Yaskawa INFORM job: A_ROOF_UPPER_0614_2_PAINT_20.JBI

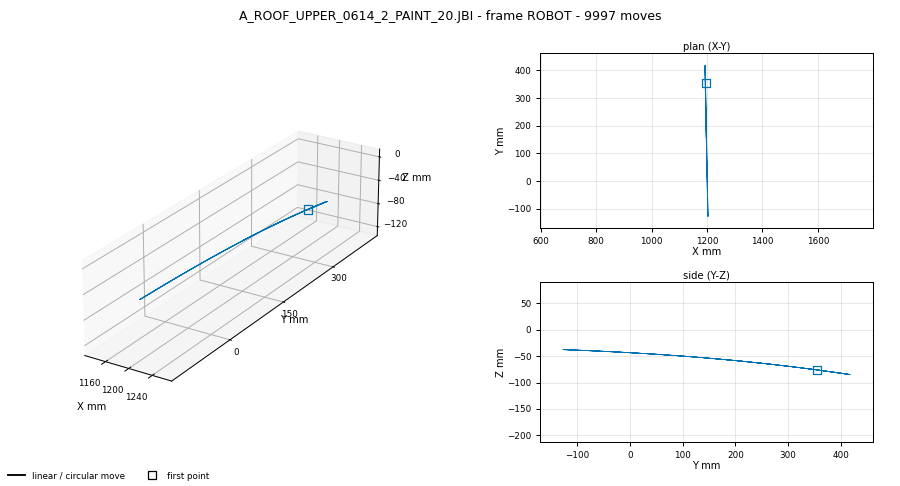
[picture p0: tool path of A_ROOF_UPPER_0614_2_PAINT_20.JBI in frame ROBOT, 9997 of 9997 moves have a stored position in this frame; points joined in program order, loops and branches not executed]
/JOB
//NAME A_ROOF_UPPER_0614_2_PAINT20
//POS
///NPOS 9997,0,0,0,0,0
///TOOL 1
///USER 0
///POSTYPE ROBOT
///RECTAN
///RCONF 1,0,0,0,0,0,0,0,0,0,0,0,0,0,0,0,0,0,0,0,0,0,0,0
C00000=1195.364,354.255,-75.937,-176.133,8.078,148.451
C00001=1195.360,354.502,-75.970,-176.131,8.082,148.451
C00002=1195.356,354.750,-76.004,-176.129,8.085,148.451
C00003=1195.352,354.998,-76.037,-176.128,8.088,148.452
C00004=1195.347,355.246,-76.070,-176.126,8.091,148.452
C00005=1195.343,355.493,-76.103,-176.124,8.095,148.452
C00006=1195.339,355.741,-76.136,-176.122,8.098,148.452
C00007=1195.335,355.989,-76.169,-176.120,8.101,148.453
C00008=1195.331,356.236,-76.203,-176.118,8.104,148.453
C00009=1195.327,356.484,-76.236,-176.116,8.107,148.453
C00010=1195.323,356.732,-76.269,-176.114,8.111,148.454
C00011=1195.319,356.980,-76.302,-176.112,8.114,148.454
C00012=1195.315,357.227,-76.336,-176.110,8.117,148.454
C00013=1195.310,357.475,-76.370,-176.108,8.121,148.455
C00014=1195.306,357.723,-76.403,-176.106,8.124,148.455
C00015=1195.302,357.971,-76.436,-176.105,8.127,148.455
C00016=1195.298,358.219,-76.469,-176.103,8.130,148.455
C00017=1195.294,358.466,-76.503,-176.101,8.134,148.456
C00018=1195.290,358.713,-76.537,-176.099,8.137,148.456
C00019=1195.286,358.961,-76.570,-176.097,8.140,148.456
C00020=1195.282,359.210,-76.603,-176.095,8.143,148.457
C00021=1195.278,359.457,-76.636,-176.093,8.147,148.457
C00022=1195.274,359.705,-76.671,-176.091,8.150,148.457
C00023=1195.269,359.953,-76.704,-176.090,8.153,148.458
C00024=1195.265,360.200,-76.737,-176.088,8.156,148.458
C00025=1195.261,360.448,-76.770,-176.086,8.160,148.458
C00026=1195.258,360.696,-76.805,-176.084,8.163,148.459
C00027=1195.254,360.944,-76.838,-176.082,8.166,148.459
C00028=1195.249,361.192,-76.871,-176.081,8.170,148.459
C00029=1195.245,361.439,-76.905,-176.078,8.173,148.460
C00030=1195.241,361.686,-76.938,-176.077,8.176,148.460
C00031=1195.237,361.934,-76.972,-176.075,8.179,148.460
C00032=1195.234,362.182,-77.006,-176.073,8.183,148.461
C00033=1195.229,362.430,-77.040,-176.072,8.186,148.461
C00034=1195.225,362.677,-77.073,-176.070,8.189,148.461
C00035=1195.221,362.925,-77.107,-176.068,8.193,148.462
C00036=1195.217,363.173,-77.140,-176.067,8.195,148.462
C00037=1195.213,363.420,-77.174,-176.065,8.199,148.463
C00038=1195.208,363.668,-77.208,-176.063,8.202,148.463
C00039=1195.205,363.916,-77.242,-176.061,8.205,148.463
C00040=1195.201,364.163,-77.275,-176.060,8.209,148.464
C00041=1195.196,364.411,-77.309,-176.058,8.212,148.464
C00042=1195.192,364.659,-77.343,-176.056,8.215,148.464
C00043=1195.189,364.906,-77.377,-176.054,8.219,148.465
C00044=1195.184,365.154,-77.410,-176.053,8.221,148.465
C00045=1195.180,365.401,-77.444,-176.051,8.225,148.465
C00046=1195.176,365.650,-77.478,-176.050,8.229,148.466
C00047=1195.172,365.897,-77.512,-176.048,8.231,148.466
C00048=1195.167,366.178,-77.549,-176.047,8.235,148.467
C00049=1195.163,366.459,-77.588,-176.045,8.239,148.467
C00050=1195.159,366.740,-77.627,-176.043,8.242,148.468
C00051=1195.154,367.021,-77.665,-176.041,8.246,148.468
C00052=1195.150,367.268,-77.698,-176.039,8.250,148.468
C00053=1195.146,367.517,-77.733,-176.037,8.253,148.469
C00054=1195.142,367.764,-77.767,-176.036,8.256,148.469
C00055=1195.137,368.012,-77.801,-176.034,8.259,148.470
C00056=1195.133,368.259,-77.835,-176.033,8.262,148.470
C00057=1195.130,368.507,-77.869,-176.031,8.266,148.470
C00058=1195.125,368.755,-77.903,-176.030,8.269,148.471
C00059=1195.121,369.002,-77.937,-176.028,8.272,148.471
C00060=1195.117,369.250,-77.971,-176.027,8.275,148.472
C00061=1195.113,369.498,-78.005,-176.025,8.279,148.472
C00062=1195.109,369.745,-78.038,-176.024,8.282,148.473
C00063=1195.105,369.993,-78.073,-176.023,8.285,148.473
C00064=1195.101,370.241,-78.106,-176.021,8.288,148.473
C00065=1195.097,370.488,-78.141,-176.020,8.292,148.474
C00066=1195.093,370.735,-78.175,-176.018,8.295,148.474
C00067=1195.089,370.983,-78.210,-176.017,8.297,148.475
C00068=1195.085,371.231,-78.243,-176.015,8.301,148.475
C00069=1195.080,371.478,-78.277,-176.014,8.304,148.475
C00070=1195.077,371.726,-78.312,-176.012,8.307,148.476
C00071=1195.073,371.973,-78.345,-176.012,8.311,148.476
C00072=1195.069,372.221,-78.380,-176.010,8.314,148.477
C00073=1195.065,372.469,-78.413,-176.009,8.317,148.477
C00074=1195.060,372.717,-78.448,-176.007,8.320,148.478
C00075=1195.057,372.964,-78.482,-176.005,8.323,148.478
C00076=1195.053,373.212,-78.517,-176.005,8.327,148.479
C00077=1195.048,373.459,-78.551,-176.003,8.329,148.479
C00078=1195.045,373.707,-78.585,-176.002,8.333,148.480
C00079=1195.040,373.955,-78.619,-176.001,8.336,148.480
C00080=1195.036,374.202,-78.653,-175.999,8.340,148.481
C00081=1195.032,374.450,-78.688,-175.998,8.343,148.481
C00082=1195.028,374.697,-78.722,-175.997,8.345,148.481
C00083=1195.024,374.945,-78.756,-175.996,8.348,148.482
C00084=1195.020,375.193,-78.790,-175.994,8.352,148.482
C00085=1195.016,375.440,-78.825,-175.993,8.355,148.483
C00086=1195.013,375.688,-78.859,-175.992,8.358,148.483
C00087=1195.008,375.935,-78.893,-175.990,8.362,148.484
C00088=1195.004,376.183,-78.928,-175.989,8.365,148.484
C00089=1195.000,376.430,-78.962,-175.988,8.367,148.485
C00090=1194.996,376.678,-78.997,-175.987,8.370,148.485
C00091=1194.992,376.926,-79.031,-175.986,8.374,148.486
C00092=1194.988,377.173,-79.065,-175.984,8.377,148.486
C00093=1194.984,377.421,-79.100,-175.984,8.380,148.487
C00094=1194.980,377.668,-79.134,-175.982,8.383,148.487
C00095=1194.976,377.916,-79.168,-175.981,8.387,148.488
C00096=1194.972,378.164,-79.203,-175.980,8.390,148.488
C00097=1194.968,378.411,-79.237,-175.979,8.393,148.489
C00098=1194.964,378.659,-79.272,-175.978,8.396,148.489
C00099=1194.960,378.906,-79.306,-175.977,8.399,148.490
C00100=1194.956,379.154,-79.341,-175.976,8.401,148.490
C00101=1194.951,379.402,-79.375,-175.974,8.405,148.491
C00102=1194.948,379.650,-79.409,-175.973,8.408,148.491
C00103=1194.944,379.897,-79.444,-175.972,8.411,148.492
C00104=1194.939,380.144,-79.478,-175.972,8.414,148.492
C00105=1194.935,380.393,-79.513,-175.970,8.417,148.493
C00106=1194.932,380.639,-79.548,-175.970,8.420,148.493
C00107=1194.928,380.887,-79.583,-175.968,8.423,148.494
C00108=1194.923,381.135,-79.617,-175.968,8.426,148.494
C00109=1194.920,381.382,-79.651,-175.967,8.429,148.495
C00110=1194.915,381.630,-79.686,-175.966,8.432,148.495
C00111=1194.911,381.878,-79.721,-175.965,8.435,148.496
C00112=1194.907,382.125,-79.755,-175.964,8.438,148.496
C00113=1194.904,382.373,-79.790,-175.963,8.441,148.497
C00114=1194.899,382.620,-79.825,-175.962,8.444,148.497
C00115=1194.895,382.868,-79.859,-175.961,8.447,148.498
C00116=1194.891,383.115,-79.893,-175.960,8.450,148.499
C00117=1194.887,383.363,-79.928,-175.959,8.453,148.499
C00118=1194.883,383.610,-79.963,-175.958,8.456,148.500
C00119=1194.879,383.858,-79.998,-175.958,8.459,148.500
C00120=1194.875,384.105,-80.032,-175.957,8.463,148.501
C00121=1194.871,384.353,-80.067,-175.956,8.465,148.501
C00122=1194.867,384.600,-80.102,-175.955,8.468,148.502
C00123=1194.863,384.848,-80.137,-175.954,8.472,148.502
C00124=1194.859,385.096,-80.171,-175.953,8.475,148.503
C00125=1194.855,385.344,-80.205,-175.953,8.477,148.503
C00126=1194.851,385.590,-80.241,-175.952,8.480,148.504
C00127=1194.847,385.839,-80.275,-175.951,8.483,148.504
C00128=1194.843,386.086,-80.310,-175.950,8.486,148.505
C00129=1194.839,386.333,-80.346,-175.949,8.489,148.506
C00130=1194.835,386.581,-80.379,-175.949,8.492,148.506
C00131=1194.831,386.829,-80.414,-175.948,8.494,148.507
C00132=1194.827,387.075,-80.449,-175.948,8.497,148.507
C00133=1194.823,387.324,-80.484,-175.947,8.501,148.508
C00134=1194.819,387.572,-80.519,-175.946,8.503,148.508
C00135=1194.815,387.819,-80.554,-175.945,8.506,148.509
C00136=1194.811,388.066,-80.588,-175.945,8.509,148.509
C00137=1194.807,388.314,-80.623,-175.944,8.512,148.510
C00138=1194.803,388.561,-80.658,-175.943,8.515,148.511
C00139=1194.799,388.809,-80.693,-175.943,8.517,148.511
C00140=1194.795,389.056,-80.729,-175.942,8.520,148.512
C00141=1194.790,389.304,-80.763,-175.941,8.523,148.512
C00142=1194.787,389.551,-80.797,-175.941,8.526,148.513
C00143=1194.783,389.799,-80.833,-175.940,8.529,148.513
C00144=1194.779,390.046,-80.867,-175.940,8.531,148.514
C00145=1194.775,390.294,-80.903,-175.939,8.534,148.514
C00146=1194.771,390.541,-80.937,-175.938,8.537,148.515
C00147=1194.767,390.789,-80.973,-175.938,8.539,148.516
C00148=1194.762,391.036,-81.007,-175.937,8.543,148.516
C00149=1194.758,391.284,-81.042,-175.937,8.545,148.517
C00150=1194.755,391.532,-81.078,-175.936,8.548,148.517
C00151=1194.751,391.779,-81.112,-175.936,8.550,148.518
C00152=1194.747,392.062,-81.152,-175.935,8.553,148.518
C00153=1194.741,392.346,-81.192,-175.934,8.556,148.519
C00154=1194.738,392.629,-81.232,-175.934,8.560,148.520
C00155=1194.732,392.912,-81.272,-175.933,8.563,148.520
C00156=1194.729,393.159,-81.307,-175.933,8.565,148.521
C00157=1194.724,393.407,-81.342,-175.932,8.568,148.522
C00158=1194.720,393.654,-81.377,-175.932,8.571,148.522
C00159=1194.717,393.902,-81.413,-175.931,8.574,148.523
C00160=1194.713,394.149,-81.447,-175.931,8.576,148.523
C00161=1194.709,394.396,-81.482,-175.930,8.579,148.524
C00162=1194.705,394.645,-81.517,-175.930,8.581,148.524
C00163=1194.701,394.891,-81.552,-175.930,8.584,148.525
C00164=1194.697,395.139,-81.587,-175.929,8.587,148.526
C00165=1194.693,395.386,-81.622,-175.929,8.589,148.526
C00166=1194.689,395.634,-81.657,-175.928,8.592,148.527
C00167=1194.685,395.882,-81.693,-175.928,8.595,148.527
C00168=1194.681,396.129,-81.728,-175.928,8.597,148.528
C00169=1194.677,396.377,-81.763,-175.927,8.600,148.528
C00170=1194.673,396.624,-81.798,-175.927,8.602,148.529
C00171=1194.669,396.872,-81.833,-175.927,8.604,148.529
C00172=1194.665,397.119,-81.868,-175.926,8.608,148.530
C00173=1194.661,397.366,-81.904,-175.926,8.610,148.531
C00174=1194.657,397.614,-81.938,-175.925,8.612,148.531
C00175=1194.653,397.862,-81.974,-175.925,8.615,148.532
C00176=1194.648,398.109,-82.008,-175.924,8.617,148.532
C00177=1194.645,398.357,-82.044,-175.924,8.620,148.533
C00178=1194.641,398.604,-82.080,-175.924,8.622,148.533
C00179=1194.637,398.851,-82.114,-175.924,8.625,148.534
C00180=1194.633,399.099,-82.150,-175.923,8.628,148.535
C00181=1194.629,399.346,-82.185,-175.923,8.630,148.535
C00182=1194.625,399.594,-82.220,-175.923,8.632,148.536
C00183=1194.621,399.841,-82.255,-175.923,8.635,148.536
C00184=1194.617,400.089,-82.291,-175.922,8.638,148.537
C00185=1194.613,400.336,-82.325,-175.922,8.640,148.537
C00186=1194.609,400.584,-82.361,-175.921,8.642,148.538
C00187=1194.605,400.831,-82.396,-175.921,8.644,148.538
C00188=1194.601,401.079,-82.431,-175.921,8.647,148.539
C00189=1194.596,401.327,-82.467,-175.921,8.649,148.539
C00190=1194.593,401.574,-82.502,-175.920,8.652,148.540
C00191=1194.588,401.821,-82.537,-175.920,8.655,148.541
C00192=1194.585,402.069,-82.572,-175.920,8.657,148.541
C00193=1194.581,402.316,-82.608,-175.920,8.659,148.542
C00194=1194.577,402.563,-82.643,-175.919,8.661,148.542
C00195=1194.573,402.811,-82.678,-175.919,8.664,148.543
C00196=1194.569,403.059,-82.713,-175.919,8.666,148.543
C00197=1194.565,403.306,-82.749,-175.919,8.668,148.544
C00198=1194.561,403.553,-82.784,-175.918,8.670,148.544
C00199=1194.557,403.801,-82.819,-175.918,8.673,148.545
C00200=1194.553,404.048,-82.854,-175.917,8.676,148.545
C00201=1194.549,404.296,-82.890,-175.917,8.678,148.546
C00202=1194.546,404.543,-82.925,-175.917,8.680,148.547
C00203=1194.541,404.792,-82.961,-175.917,8.683,148.547
C00204=1194.537,405.038,-82.996,-175.917,8.685,148.548
C00205=1194.533,405.286,-83.031,-175.917,8.687,148.548
C00206=1194.529,405.533,-83.067,-175.916,8.690,148.549
C00207=1194.525,405.781,-83.101,-175.916,8.692,148.549
C00208=1194.521,406.028,-83.137,-175.916,8.694,148.550
C00209=1194.517,406.276,-83.173,-175.916,8.697,148.550
C00210=1194.513,406.523,-83.208,-175.915,8.699,148.551
C00211=1194.509,406.770,-83.243,-175.915,8.701,148.551
C00212=1194.505,407.019,-83.279,-175.915,8.703,148.552
C00213=1194.501,407.266,-83.314,-175.915,8.706,148.553
C00214=1194.497,407.513,-83.349,-175.914,8.708,148.553
C00215=1194.493,407.760,-83.385,-175.914,8.710,148.554
C00216=1194.489,408.008,-83.421,-175.914,8.712,148.554
C00217=1194.485,408.255,-83.456,-175.914,8.714,148.555
C00218=1194.481,408.503,-83.491,-175.914,8.716,148.555
C00219=1194.478,408.750,-83.526,-175.914,8.718,148.556
C00220=1194.473,408.998,-83.562,-175.913,8.721,148.556
C00221=1194.469,409.245,-83.597,-175.913,8.723,148.557
C00222=1194.465,409.492,-83.633,-175.913,8.725,148.557
C00223=1194.462,409.740,-83.669,-175.913,8.727,148.558
C00224=1194.458,409.987,-83.704,-175.913,8.730,148.558
C00225=1194.453,410.235,-83.739,-175.912,8.732,148.559
C00226=1194.450,410.482,-83.774,-175.913,8.733,148.559
C00227=1194.445,410.730,-83.810,-175.912,8.736,148.560
C00228=1194.442,410.978,-83.846,-175.912,8.738,148.560
C00229=1194.437,411.224,-83.881,-175.912,8.740,148.561
C00230=1194.434,411.472,-83.917,-175.912,8.742,148.561
C00231=1194.430,411.719,-83.952,-175.911,8.745,148.562
C00232=1194.426,411.967,-83.988,-175.911,8.747,148.562
C00233=1194.421,412.214,-84.023,-175.911,8.748,148.563
C00234=1194.418,412.461,-84.059,-175.911,8.751,148.563
C00235=1194.414,412.710,-84.094,-175.911,8.753,148.564
C00236=1194.410,412.957,-84.129,-175.911,8.755,148.564
C00237=1194.406,413.204,-84.165,-175.910,8.757,148.565
C00238=1194.401,413.452,-84.201,-175.910,8.760,148.566
C00239=1194.398,413.699,-84.236,-175.911,8.761,148.566
C00240=1194.394,413.947,-84.272,-175.910,8.763,148.567
C00241=1194.390,414.194,-84.307,-175.910,8.766,148.567
C00242=1194.386,414.441,-84.342,-175.910,8.768,148.568
C00243=1194.382,414.689,-84.379,-175.910,8.769,148.568
C00244=1194.378,414.936,-84.414,-175.909,8.771,148.568
C00245=1194.374,415.183,-84.449,-175.909,8.774,148.569
C00246=1194.370,415.431,-84.485,-175.909,8.776,148.569
C00247=1194.367,415.678,-84.520,-175.909,8.778,148.570
C00248=1194.360,416.037,-84.572,-175.909,8.781,148.571
C00249=1194.357,416.395,-84.624,-175.909,8.784,148.571
C00250=1194.356,416.753,-84.674,-175.908,8.786,148.572
C00251=1194.359,417.111,-84.725,-175.908,8.789,148.573
C00252=1193.937,417.112,-84.765,-175.912,8.800,148.576
C00253=1193.935,416.751,-84.714,-175.911,8.797,148.576
C00254=1193.935,416.390,-84.662,-175.912,8.795,148.575
C00255=1193.939,416.028,-84.610,-175.912,8.791,148.574
C00256=1193.945,415.668,-84.558,-175.912,8.789,148.574
C00257=1193.949,415.420,-84.523,-175.912,8.787,148.573
C00258=1193.952,415.173,-84.487,-175.912,8.784,148.573
C00259=1193.956,414.925,-84.452,-175.913,8.782,148.572
C00260=1193.961,414.678,-84.416,-175.912,8.781,148.572
C00261=1193.965,414.431,-84.381,-175.913,8.779,148.571
C00262=1193.968,414.183,-84.345,-175.913,8.776,148.571
C00263=1193.972,413.935,-84.310,-175.913,8.774,148.570
C00264=1193.976,413.688,-84.275,-175.914,8.772,148.570
C00265=1193.981,413.440,-84.239,-175.913,8.770,148.569
C00266=1193.985,413.193,-84.203,-175.914,8.768,148.569
C00267=1193.988,412.945,-84.168,-175.914,8.766,148.568
C00268=1193.992,412.698,-84.132,-175.914,8.764,148.568
C00269=1193.996,412.451,-84.097,-175.914,8.761,148.567
C00270=1194.001,412.203,-84.061,-175.914,8.760,148.567
C00271=1194.004,411.956,-84.025,-175.914,8.758,148.566
C00272=1194.008,411.708,-83.990,-175.915,8.755,148.566
C00273=1194.012,411.462,-83.955,-175.915,8.753,148.565
C00274=1194.016,411.214,-83.919,-175.915,8.751,148.565
C00275=1194.020,410.966,-83.883,-175.915,8.749,148.564
C00276=1194.024,410.718,-83.848,-175.915,8.746,148.563
C00277=1194.028,410.471,-83.813,-175.915,8.745,148.563
C00278=1194.032,410.224,-83.777,-175.915,8.743,148.562
C00279=1194.036,409.976,-83.742,-175.916,8.740,148.562
C00280=1194.039,409.729,-83.706,-175.916,8.738,148.561
C00281=1194.044,409.482,-83.670,-175.916,8.736,148.561
C00282=1194.048,409.234,-83.635,-175.916,8.734,148.560
C00283=1194.052,408.987,-83.599,-175.917,8.731,148.560
C00284=1194.055,408.739,-83.564,-175.917,8.729,148.559
C00285=1194.060,408.492,-83.529,-175.917,8.728,148.559
C00286=1194.064,408.244,-83.494,-175.917,8.725,148.558
C00287=1194.067,407.997,-83.458,-175.917,8.723,148.558
C00288=1194.072,407.750,-83.422,-175.917,8.721,148.557
C00289=1194.076,407.502,-83.387,-175.918,8.719,148.557
C00290=1194.080,407.255,-83.351,-175.918,8.716,148.556
C00291=1194.084,407.007,-83.317,-175.918,8.714,148.556
C00292=1194.088,406.760,-83.281,-175.918,8.712,148.555
C00293=1194.091,406.512,-83.246,-175.918,8.709,148.555
C00294=1194.095,406.265,-83.210,-175.918,8.707,148.554
C00295=1194.099,406.018,-83.175,-175.919,8.705,148.553
C00296=1194.104,405.770,-83.139,-175.919,8.702,148.553
C00297=1194.108,405.522,-83.104,-175.919,8.700,148.552
C00298=1194.111,405.274,-83.069,-175.919,8.698,148.552
C00299=1194.116,405.028,-83.033,-175.919,8.696,148.551
C00300=1194.119,404.780,-82.998,-175.920,8.693,148.551
C00301=1194.123,404.532,-82.963,-175.920,8.691,148.550
C00302=1194.128,404.285,-82.928,-175.920,8.689,148.550
C00303=1194.131,404.038,-82.892,-175.920,8.686,148.549
C00304=1194.135,403.790,-82.857,-175.921,8.684,148.549
C00305=1194.139,403.543,-82.821,-175.921,8.682,148.548
C00306=1194.144,403.295,-82.786,-175.921,8.680,148.548
C00307=1194.148,403.048,-82.751,-175.921,8.677,148.547
C00308=1194.151,402.800,-82.715,-175.921,8.675,148.546
C00309=1194.156,402.553,-82.680,-175.922,8.672,148.546
C00310=1194.159,402.305,-82.645,-175.922,8.669,148.545
C00311=1194.163,402.058,-82.609,-175.922,8.667,148.545
C00312=1194.167,401.811,-82.574,-175.923,8.665,148.544
C00313=1194.171,401.563,-82.539,-175.923,8.663,148.544
C00314=1194.175,401.315,-82.504,-175.923,8.660,148.543
C00315=1194.179,401.068,-82.469,-175.923,8.658,148.543
C00316=1194.183,400.821,-82.433,-175.924,8.656,148.542
C00317=1194.187,400.573,-82.398,-175.924,8.653,148.541
C00318=1194.191,400.326,-82.363,-175.925,8.651,148.541
C00319=1194.195,400.078,-82.328,-175.925,8.648,148.540
C00320=1194.199,399.830,-82.293,-175.925,8.646,148.540
C00321=1194.203,399.584,-82.258,-175.925,8.643,148.539
C00322=1194.207,399.336,-82.222,-175.926,8.640,148.539
C00323=1194.211,399.088,-82.187,-175.926,8.638,148.538
C00324=1194.215,398.841,-82.152,-175.926,8.636,148.537
C00325=1194.219,398.593,-82.116,-175.927,8.634,148.537
C00326=1194.223,398.345,-82.081,-175.927,8.630,148.536
C00327=1194.228,398.098,-82.046,-175.928,8.628,148.536
C00328=1194.231,397.851,-82.010,-175.928,8.626,148.535
C00329=1194.235,397.603,-81.975,-175.928,8.623,148.535
C00330=1194.240,397.356,-81.940,-175.928,8.620,148.534
C00331=1194.243,397.108,-81.905,-175.929,8.618,148.533
C00332=1194.248,396.861,-81.870,-175.929,8.616,148.533
C00333=1194.251,396.614,-81.835,-175.930,8.613,148.532
C00334=1194.255,396.365,-81.800,-175.930,8.610,148.532
C00335=1194.260,396.119,-81.765,-175.930,8.608,148.531
C00336=1194.264,395.871,-81.730,-175.931,8.605,148.531
C00337=1194.267,395.623,-81.694,-175.931,8.603,148.530
C00338=1194.272,395.376,-81.659,-175.931,8.600,148.530
C00339=1194.275,395.128,-81.624,-175.932,8.597,148.529
C00340=1194.278,394.881,-81.589,-175.932,8.595,148.529
C00341=1194.283,394.633,-81.555,-175.932,8.592,148.528
C00342=1194.287,394.386,-81.519,-175.933,8.589,148.527
C00343=1194.291,394.139,-81.485,-175.933,8.587,148.527
C00344=1194.295,393.891,-81.449,-175.934,8.584,148.526
C00345=1194.299,393.644,-81.414,-175.934,8.582,148.526
C00346=1194.303,393.396,-81.379,-175.935,8.579,148.525
C00347=1194.307,393.149,-81.344,-175.935,8.576,148.524
C00348=1194.311,392.901,-81.309,-175.936,8.573,148.524
C00349=1194.316,392.618,-81.269,-175.936,8.571,148.523
C00350=1194.320,392.334,-81.229,-175.937,8.568,148.523
C00351=1194.325,392.052,-81.189,-175.937,8.565,148.522
C00352=1194.330,391.768,-81.149,-175.938,8.561,148.521
C00353=1194.333,391.521,-81.114,-175.939,8.558,148.521
C00354=1194.337,391.273,-81.079,-175.939,8.556,148.520
C00355=1194.341,391.026,-81.044,-175.940,8.553,148.520
C00356=1194.345,390.778,-81.009,-175.940,8.551,148.519
C00357=1194.349,390.530,-80.974,-175.941,8.548,148.519
C00358=1194.353,390.283,-80.939,-175.941,8.545,148.518
C00359=1194.357,390.035,-80.904,-175.942,8.542,148.517
C00360=1194.362,389.788,-80.869,-175.943,8.539,148.517
C00361=1194.366,389.540,-80.834,-175.943,8.537,148.516
C00362=1194.369,389.294,-80.800,-175.944,8.534,148.516
C00363=1194.373,389.045,-80.765,-175.945,8.531,148.515
C00364=1194.377,388.798,-80.729,-175.945,8.528,148.515
C00365=1194.381,388.550,-80.695,-175.946,8.525,148.514
C00366=1194.385,388.302,-80.660,-175.947,8.522,148.513
C00367=1194.390,388.056,-80.625,-175.947,8.520,148.513
C00368=1194.394,387.807,-80.590,-175.948,8.517,148.512
C00369=1194.397,387.560,-80.556,-175.948,8.514,148.512
C00370=1194.401,387.313,-80.521,-175.949,8.511,148.511
C00371=1194.405,387.065,-80.486,-175.949,8.508,148.511
C00372=1194.409,386.818,-80.451,-175.950,8.505,148.510
C00373=1194.413,386.570,-80.416,-175.951,8.502,148.510
C00374=1194.418,386.322,-80.381,-175.952,8.499,148.509
C00375=1194.421,386.075,-80.346,-175.953,8.496,148.508
C00376=1194.425,385.828,-80.312,-175.953,8.494,148.508
C00377=1194.429,385.580,-80.277,-175.954,8.491,148.507
C00378=1194.434,385.332,-80.243,-175.955,8.488,148.507
C00379=1194.438,385.085,-80.207,-175.956,8.485,148.506
C00380=1194.441,384.838,-80.173,-175.957,8.482,148.506
C00381=1194.445,384.590,-80.138,-175.958,8.479,148.505
C00382=1194.450,384.343,-80.103,-175.958,8.476,148.505
C00383=1194.454,384.095,-80.068,-175.959,8.473,148.504
C00384=1194.457,383.847,-80.034,-175.959,8.470,148.503
C00385=1194.461,383.599,-80.000,-175.961,8.468,148.503
C00386=1194.466,383.353,-79.964,-175.961,8.464,148.503
C00387=1194.470,383.104,-79.930,-175.962,8.461,148.502
C00388=1194.473,382.857,-79.896,-175.963,8.458,148.501
C00389=1194.477,382.609,-79.861,-175.964,8.455,148.501
C00390=1194.482,382.362,-79.826,-175.965,8.452,148.500
C00391=1194.486,382.114,-79.791,-175.966,8.449,148.500
C00392=1194.489,381.867,-79.757,-175.967,8.446,148.499
C00393=1194.493,381.619,-79.722,-175.968,8.443,148.499
C00394=1194.498,381.372,-79.688,-175.969,8.440,148.498
C00395=1194.502,381.124,-79.653,-175.970,8.437,148.498
C00396=1194.506,380.876,-79.619,-175.971,8.434,148.497
C00397=1194.509,380.629,-79.583,-175.972,8.430,148.497
C00398=1194.514,380.381,-79.549,-175.973,8.428,148.496
C00399=1194.517,380.134,-79.515,-175.974,8.424,148.496
C00400=1194.522,379.886,-79.480,-175.975,8.421,148.495
C00401=1194.526,379.638,-79.445,-175.976,8.419,148.495
C00402=1194.530,379.391,-79.412,-175.977,8.415,148.494
C00403=1194.534,379.144,-79.377,-175.978,8.413,148.494
C00404=1194.538,378.895,-79.342,-175.979,8.410,148.493
C00405=1194.543,378.648,-79.308,-175.981,8.406,148.493
C00406=1194.546,378.400,-79.274,-175.981,8.403,148.492
C00407=1194.550,378.153,-79.238,-175.983,8.400,148.492
C00408=1194.553,377.906,-79.204,-175.983,8.397,148.491
C00409=1194.558,377.658,-79.170,-175.985,8.394,148.491
C00410=1194.563,377.411,-79.135,-175.986,8.390,148.490
C00411=1194.566,377.163,-79.101,-175.987,8.387,148.490
C00412=1194.570,376.916,-79.066,-175.988,8.384,148.489
C00413=1194.574,376.667,-79.032,-175.989,8.381,148.489
C00414=1194.578,376.420,-78.998,-175.990,8.378,148.488
C00415=1194.582,376.172,-78.963,-175.992,8.375,148.488
C00416=1194.586,375.925,-78.929,-175.993,8.372,148.487
C00417=1194.591,375.678,-78.895,-175.994,8.369,148.487
C00418=1194.595,375.430,-78.860,-175.996,8.365,148.486
C00419=1194.599,375.182,-78.827,-175.996,8.362,148.486
C00420=1194.603,374.934,-78.792,-175.998,8.359,148.485
C00421=1194.607,374.687,-78.758,-175.999,8.356,148.485
C00422=1194.611,374.439,-78.723,-176.000,8.353,148.484
C00423=1194.614,374.191,-78.689,-176.001,8.350,148.484
C00424=1194.619,373.944,-78.655,-176.003,8.346,148.483
C00425=1194.622,373.696,-78.621,-176.004,8.343,148.483
C00426=1194.627,373.449,-78.586,-176.005,8.340,148.482
C00427=1194.631,373.202,-78.552,-176.007,8.337,148.482
C00428=1194.634,372.954,-78.517,-176.008,8.334,148.482
C00429=1194.639,372.705,-78.484,-176.009,8.331,148.481
C00430=1194.643,372.458,-78.450,-176.011,8.327,148.481
C00431=1194.647,372.210,-78.415,-176.012,8.324,148.480
C00432=1194.651,371.963,-78.381,-176.014,8.321,148.480
C00433=1194.656,371.716,-78.347,-176.015,8.318,148.479
C00434=1194.659,371.467,-78.313,-176.016,8.315,148.479
C00435=1194.663,371.220,-78.279,-176.018,8.311,148.478
C00436=1194.667,370.973,-78.245,-176.019,8.308,148.478
C00437=1194.671,370.725,-78.210,-176.021,8.305,148.478
C00438=1194.675,370.478,-78.176,-176.022,8.302,148.477
C00439=1194.679,370.230,-78.143,-176.024,8.298,148.477
C00440=1194.683,369.982,-78.108,-176.025,8.295,148.476
C00441=1194.687,369.735,-78.074,-176.027,8.292,148.476
C00442=1194.692,369.487,-78.040,-176.028,8.289,148.476
C00443=1194.695,369.239,-78.006,-176.030,8.285,148.475
C00444=1194.700,368.991,-77.972,-176.031,8.283,148.475
C00445=1194.704,368.744,-77.938,-176.032,8.279,148.474
C00446=1194.707,368.496,-77.904,-176.034,8.276,148.474
C00447=1194.712,368.248,-77.870,-176.035,8.272,148.473
C00448=1194.716,368.001,-77.837,-176.037,8.269,148.473
C00449=1194.721,367.753,-77.802,-176.039,8.266,148.473
C00450=1194.724,367.505,-77.768,-176.040,8.263,148.472
C00451=1194.728,367.258,-77.735,-176.042,8.260,148.472
C00452=1194.733,367.010,-77.700,-176.044,8.256,148.471
C00453=1194.737,366.729,-77.661,-176.045,8.252,148.471
C00454=1194.741,366.448,-77.623,-176.047,8.249,148.470
C00455=1194.746,366.167,-77.585,-176.049,8.245,148.470
C00456=1194.750,365.887,-77.547,-176.051,8.241,148.470
C00457=1194.754,365.639,-77.512,-176.052,8.239,148.469
C00458=1194.759,365.391,-77.479,-176.054,8.235,148.469
C00459=1194.762,365.144,-77.445,-176.056,8.231,148.468
C00460=1194.767,364.896,-77.412,-176.057,8.229,148.468
C00461=1194.770,364.648,-77.377,-176.059,8.225,148.468
C00462=1194.775,364.400,-77.344,-176.060,8.222,148.467
C00463=1194.779,364.153,-77.310,-176.062,8.219,148.467
C00464=1194.783,363.905,-77.277,-176.064,8.215,148.466
C00465=1194.787,363.657,-77.242,-176.065,8.212,148.466
C00466=1194.791,363.410,-77.209,-176.067,8.209,148.466
C00467=1194.795,363.162,-77.175,-176.069,8.205,148.465
C00468=1194.799,362.914,-77.142,-176.070,8.203,148.465
C00469=1194.804,362.667,-77.109,-176.073,8.199,148.465
C00470=1194.807,362.419,-77.074,-176.074,8.196,148.464
C00471=1194.811,362.171,-77.041,-176.076,8.193,148.464
C00472=1194.815,361.924,-77.007,-176.077,8.189,148.464
C00473=1194.820,361.676,-76.974,-176.080,8.186,148.463
C00474=1194.824,361.428,-76.940,-176.081,8.183,148.463
C00475=1194.827,361.180,-76.906,-176.083,8.180,148.463
C00476=1194.831,360.933,-76.873,-176.085,8.176,148.462
C00477=1194.836,360.685,-76.839,-176.087,8.173,148.462
C00478=1194.840,360.438,-76.805,-176.088,8.170,148.462
C00479=1194.844,360.190,-76.772,-176.090,8.166,148.461
C00480=1194.848,359.942,-76.739,-176.092,8.163,148.461
C00481=1194.852,359.694,-76.706,-176.094,8.159,148.461
C00482=1194.855,359.447,-76.672,-176.096,8.157,148.460
C00483=1194.860,359.199,-76.638,-176.098,8.153,148.460
C00484=1194.864,358.951,-76.605,-176.100,8.150,148.460
C00485=1194.869,358.703,-76.572,-176.101,8.147,148.459
C00486=1194.872,358.456,-76.538,-176.103,8.144,148.459
C00487=1194.877,358.208,-76.505,-176.105,8.140,148.459
C00488=1194.880,357.960,-76.471,-176.107,8.137,148.458
C00489=1194.884,357.712,-76.438,-176.109,8.133,148.458
C00490=1194.888,357.464,-76.405,-176.111,8.131,148.458
C00491=1194.892,357.217,-76.371,-176.113,8.127,148.457
C00492=1194.897,356.969,-76.337,-176.115,8.124,148.457
C00493=1194.901,356.721,-76.304,-176.117,8.120,148.457
C00494=1194.905,356.474,-76.271,-176.118,8.118,148.457
C00495=1194.910,356.226,-76.238,-176.120,8.114,148.456
C00496=1194.914,355.978,-76.204,-176.122,8.111,148.456
C00497=1194.918,355.731,-76.171,-176.125,8.107,148.456
C00498=1194.921,355.482,-76.138,-176.126,8.105,148.455
C00499=1194.925,355.234,-76.105,-176.128,8.101,148.455
C00500=1194.930,354.987,-76.071,-176.130,8.098,148.455
C00501=1194.934,354.739,-76.038,-176.132,8.095,148.455
C00502=1194.938,354.492,-76.004,-176.134,8.091,148.454
C00503=1194.942,354.244,-75.971,-176.136,8.088,148.454
C00504=1194.946,353.996,-75.938,-176.138,8.085,148.454
C00505=1194.950,353.749,-75.905,-176.140,8.081,148.453
C00506=1194.954,353.500,-75.873,-176.142,8.078,148.453
C00507=1194.959,353.253,-75.839,-176.144,8.076,148.453
C00508=1194.963,353.005,-75.806,-176.146,8.072,148.453
C00509=1194.967,352.757,-75.773,-176.148,8.069,148.452
C00510=1194.971,352.509,-75.740,-176.150,8.065,148.452
C00511=1194.975,352.262,-75.707,-176.152,8.062,148.452
C00512=1194.979,352.014,-75.674,-176.154,8.059,148.452
C00513=1194.983,351.766,-75.641,-176.156,8.056,148.451
C00514=1194.987,351.519,-75.608,-176.158,8.052,148.451
C00515=1194.991,351.271,-75.575,-176.160,8.049,148.451
C00516=1194.995,351.023,-75.542,-176.162,8.047,148.451
C00517=1195.000,350.775,-75.509,-176.164,8.043,148.450
C00518=1195.004,350.527,-75.476,-176.166,8.040,148.450
C00519=1195.008,350.279,-75.443,-176.168,8.036,148.450
C00520=1195.012,350.032,-75.410,-176.170,8.033,148.449
C00521=1195.016,349.784,-75.377,-176.172,8.031,148.449
C00522=1195.020,349.536,-75.345,-176.174,8.027,148.449
C00523=1195.024,349.288,-75.312,-176.177,8.024,148.449
C00524=1195.028,349.041,-75.278,-176.179,8.021,148.449
C00525=1195.032,348.793,-75.245,-176.181,8.017,148.448
C00526=1195.036,348.545,-75.212,-176.182,8.014,148.448
C00527=1195.041,348.297,-75.180,-176.184,8.011,148.448
C00528=1195.044,348.049,-75.147,-176.187,8.008,148.448
C00529=1195.048,347.802,-75.114,-176.189,8.004,148.447
C00530=1195.053,347.554,-75.082,-176.191,8.002,148.447
C00531=1195.058,347.306,-75.049,-176.193,7.999,148.447
C00532=1195.062,347.058,-75.016,-176.195,7.995,148.447
C00533=1195.065,346.810,-74.984,-176.197,7.992,148.447
C00534=1195.069,346.563,-74.951,-176.200,7.989,148.446
C00535=1195.074,346.315,-74.917,-176.201,7.986,148.446
C00536=1195.078,346.067,-74.885,-176.203,7.983,148.446
C00537=1195.081,345.819,-74.852,-176.206,7.979,148.446
C00538=1195.086,345.571,-74.820,-176.208,7.976,148.445
C00539=1195.090,345.323,-74.787,-176.210,7.973,148.445
C00540=1195.095,345.075,-74.755,-176.212,7.970,148.445
C00541=1195.098,344.828,-74.722,-176.214,7.967,148.445
C00542=1195.103,344.580,-74.689,-176.216,7.964,148.445
C00543=1195.107,344.332,-74.657,-176.219,7.960,148.444
C00544=1195.110,344.085,-74.624,-176.220,7.958,148.444
C00545=1195.115,343.836,-74.592,-176.222,7.954,148.444
C00546=1195.119,343.588,-74.558,-176.225,7.951,148.444
C00547=1195.123,343.341,-74.527,-176.227,7.948,148.444
C00548=1195.128,343.093,-74.494,-176.229,7.944,148.443
C00549=1195.132,342.845,-74.461,-176.231,7.942,148.443
C00550=1195.136,342.597,-74.429,-176.234,7.939,148.443
C00551=1195.140,342.349,-74.396,-176.236,7.936,148.443
C00552=1195.144,342.101,-74.364,-176.238,7.932,148.443
C00553=1195.148,341.854,-74.332,-176.240,7.929,148.443
C00554=1195.153,341.606,-74.299,-176.242,7.926,148.442
C00555=1195.157,341.358,-74.267,-176.244,7.923,148.442
C00556=1195.161,341.110,-74.234,-176.246,7.920,148.442
C00557=1195.165,340.832,-74.198,-176.249,7.916,148.442
C00558=1195.170,340.553,-74.162,-176.251,7.913,148.442
C00559=1195.175,340.275,-74.126,-176.254,7.909,148.441
C00560=1195.179,339.996,-74.089,-176.256,7.906,148.441
C00561=1195.184,339.748,-74.057,-176.259,7.903,148.441
C00562=1195.187,339.500,-74.024,-176.261,7.899,148.441
C00563=1195.192,339.253,-73.992,-176.263,7.897,148.441
C00564=1195.196,339.005,-73.960,-176.265,7.894,148.441
C00565=1195.200,338.756,-73.928,-176.267,7.890,148.440
C00566=1195.204,338.509,-73.895,-176.270,7.887,148.440
C00567=1195.209,338.261,-73.863,-176.271,7.885,148.440
C00568=1195.212,338.013,-73.831,-176.274,7.882,148.440
C00569=1195.217,337.765,-73.799,-176.276,7.878,148.440
C00570=1195.221,337.517,-73.767,-176.279,7.875,148.440
C00571=1195.225,337.270,-73.734,-176.281,7.872,148.439
C00572=1195.229,337.022,-73.702,-176.283,7.869,148.439
C00573=1195.234,336.773,-73.670,-176.285,7.866,148.439
C00574=1195.237,336.525,-73.638,-176.287,7.863,148.439
C00575=1195.242,336.278,-73.606,-176.290,7.859,148.439
C00576=1195.246,336.030,-73.574,-176.292,7.856,148.439
C00577=1195.250,335.781,-73.542,-176.294,7.854,148.439
C00578=1195.254,335.534,-73.509,-176.296,7.851,148.438
C00579=1195.258,335.286,-73.478,-176.298,7.847,148.438
C00580=1195.263,335.038,-73.445,-176.301,7.844,148.438
C00581=1195.266,334.790,-73.413,-176.303,7.842,148.438
C00582=1195.271,334.543,-73.382,-176.305,7.838,148.438
C00583=1195.275,334.294,-73.349,-176.308,7.835,148.438
C00584=1195.279,334.046,-73.318,-176.310,7.832,148.437
C00585=1195.284,333.799,-73.285,-176.312,7.829,148.437
C00586=1195.287,333.551,-73.254,-176.314,7.827,148.437
C00587=1195.291,333.303,-73.222,-176.317,7.823,148.437
C00588=1195.296,333.055,-73.190,-176.319,7.820,148.437
C00589=1195.300,332.807,-73.158,-176.321,7.817,148.437
C00590=1195.304,332.559,-73.126,-176.324,7.814,148.437
C00591=1195.308,332.312,-73.095,-176.325,7.811,148.436
C00592=1195.313,332.063,-73.063,-176.328,7.808,148.436
C00593=1195.317,331.815,-73.031,-176.330,7.805,148.436
C00594=1195.321,331.567,-72.999,-176.333,7.802,148.436
C00595=1195.325,331.319,-72.967,-176.335,7.799,148.436
C00596=1195.329,331.071,-72.936,-176.337,7.796,148.436
C00597=1195.333,330.823,-72.904,-176.340,7.793,148.436
C00598=1195.337,330.575,-72.872,-176.342,7.789,148.436
C00599=1195.342,330.328,-72.840,-176.345,7.786,148.436
C00600=1195.346,330.079,-72.809,-176.346,7.784,148.436
C00601=1195.350,329.832,-72.777,-176.349,7.781,148.436
C00602=1195.354,329.584,-72.745,-176.351,7.778,148.435
C00603=1195.358,329.335,-72.713,-176.353,7.774,148.435
C00604=1195.363,329.087,-72.682,-176.356,7.771,148.435
C00605=1195.367,328.839,-72.650,-176.358,7.769,148.435
C00606=1195.371,328.592,-72.619,-176.360,7.766,148.435
C00607=1195.375,328.344,-72.587,-176.363,7.762,148.435
C00608=1195.380,328.096,-72.556,-176.365,7.759,148.435
C00609=1195.384,327.848,-72.524,-176.367,7.757,148.435
C00610=1195.388,327.600,-72.492,-176.370,7.754,148.435
C00611=1195.392,327.352,-72.461,-176.372,7.751,148.434
C00612=1195.396,327.104,-72.429,-176.375,7.747,148.434
C00613=1195.400,326.856,-72.398,-176.377,7.744,148.434
C00614=1195.404,326.608,-72.367,-176.379,7.742,148.434
C00615=1195.409,326.360,-72.335,-176.381,7.739,148.434
C00616=1195.413,326.112,-72.303,-176.384,7.736,148.434
C00617=1195.417,325.864,-72.272,-176.386,7.732,148.434
C00618=1195.421,325.616,-72.240,-176.388,7.730,148.434
C00619=1195.426,325.368,-72.209,-176.391,7.727,148.434
C00620=1195.430,325.120,-72.178,-176.393,7.724,148.434
C00621=1195.434,324.873,-72.146,-176.395,7.720,148.433
C00622=1195.438,324.624,-72.115,-176.398,7.718,148.433
C00623=1195.442,324.377,-72.083,-176.400,7.715,148.433
C00624=1195.446,324.128,-72.052,-176.403,7.712,148.433
C00625=1195.450,323.881,-72.021,-176.405,7.709,148.433
C00626=1195.454,323.632,-71.990,-176.407,7.706,148.433
C00627=1195.459,323.385,-71.958,-176.410,7.703,148.433
C00628=1195.463,323.136,-71.927,-176.412,7.700,148.433
C00629=1195.467,322.889,-71.896,-176.415,7.697,148.433
C00630=1195.471,322.640,-71.864,-176.417,7.694,148.433
C00631=1195.476,322.392,-71.834,-176.419,7.691,148.433
C00632=1195.479,322.144,-71.802,-176.421,7.688,148.432
C00633=1195.484,321.896,-71.771,-176.424,7.685,148.432
C00634=1195.488,321.649,-71.740,-176.427,7.682,148.432
C00635=1195.492,321.400,-71.709,-176.428,7.680,148.432
C00636=1195.497,321.152,-71.678,-176.431,7.677,148.432
C00637=1195.501,320.904,-71.646,-176.433,7.673,148.432
C00638=1195.505,320.656,-71.615,-176.436,7.670,148.432
C00639=1195.509,320.407,-71.584,-176.439,7.667,148.432
C00640=1195.514,320.160,-71.553,-176.440,7.665,148.432
C00641=1195.518,319.912,-71.522,-176.443,7.662,148.432
C00642=1195.522,319.663,-71.491,-176.446,7.659,148.432
C00643=1195.526,319.416,-71.460,-176.448,7.655,148.432
C00644=1195.530,319.168,-71.429,-176.450,7.653,148.432
C00645=1195.534,318.920,-71.398,-176.453,7.650,148.432
C00646=1195.539,318.672,-71.367,-176.455,7.647,148.432
C00647=1195.543,318.424,-71.335,-176.458,7.644,148.432
C00648=1195.547,318.176,-71.304,-176.460,7.642,148.432
C00649=1195.551,317.927,-71.273,-176.462,7.638,148.431
C00650=1195.556,317.679,-71.243,-176.465,7.635,148.431
C00651=1195.560,317.432,-71.212,-176.467,7.632,148.431
C00652=1195.564,317.184,-71.181,-176.469,7.630,148.431
C00653=1195.568,316.936,-71.150,-176.472,7.627,148.431
C00654=1195.573,316.688,-71.119,-176.474,7.624,148.431
C00655=1195.577,316.439,-71.088,-176.477,7.620,148.431
C00656=1195.581,316.191,-71.058,-176.479,7.618,148.431
C00657=1195.585,315.943,-71.027,-176.482,7.615,148.431
C00658=1195.589,315.695,-70.996,-176.484,7.612,148.431
C00659=1195.594,315.447,-70.965,-176.486,7.609,148.431
C00660=1195.598,315.199,-70.935,-176.489,7.607,148.431
C00661=1195.603,314.922,-70.900,-176.492,7.603,148.431
C00662=1195.607,314.647,-70.865,-176.495,7.600,148.431
C00663=1195.612,314.369,-70.831,-176.497,7.596,148.431
C00664=1195.617,314.094,-70.797,-176.499,7.593,148.431
C00665=1195.621,313.846,-70.766,-176.502,7.590,148.431
C00666=1195.625,313.597,-70.736,-176.505,7.587,148.431
C00667=1195.629,313.349,-70.705,-176.507,7.585,148.431
C00668=1195.634,313.101,-70.674,-176.509,7.582,148.431
C00669=1195.638,312.854,-70.644,-176.512,7.579,148.431
C00670=1195.642,312.605,-70.613,-176.515,7.576,148.431
C00671=1195.646,312.357,-70.582,-176.516,7.573,148.431
C00672=1195.650,312.109,-70.552,-176.519,7.570,148.431
C00673=1195.655,311.861,-70.522,-176.522,7.567,148.431
C00674=1195.659,311.612,-70.491,-176.524,7.565,148.431
C00675=1195.663,311.365,-70.461,-176.527,7.562,148.431
C00676=1195.668,311.117,-70.430,-176.529,7.559,148.430
C00677=1195.672,310.869,-70.399,-176.531,7.556,148.430
C00678=1195.676,310.621,-70.369,-176.534,7.554,148.430
C00679=1195.680,310.372,-70.338,-176.536,7.551,148.430
C00680=1195.684,310.124,-70.309,-176.539,7.548,148.431
C00681=1195.689,309.876,-70.278,-176.541,7.544,148.430
C00682=1195.694,309.628,-70.247,-176.543,7.542,148.430
C00683=1195.697,309.380,-70.216,-176.546,7.539,148.430
C00684=1195.702,309.131,-70.186,-176.549,7.536,148.430
C00685=1195.706,308.884,-70.156,-176.551,7.534,148.430
C00686=1195.710,308.636,-70.125,-176.553,7.531,148.430
C00687=1195.714,308.388,-70.095,-176.556,7.527,148.430
C00688=1195.719,308.139,-70.065,-176.559,7.524,148.430
C00689=1195.722,307.891,-70.035,-176.561,7.522,148.430
C00690=1195.727,307.643,-70.004,-176.563,7.519,148.430
C00691=1195.731,307.395,-69.974,-176.566,7.516,148.430
C00692=1195.736,307.147,-69.944,-176.568,7.513,148.430
C00693=1195.740,306.899,-69.914,-176.570,7.511,148.430
C00694=1195.745,306.651,-69.884,-176.573,7.508,148.430
C00695=1195.748,306.403,-69.853,-176.576,7.505,148.430
C00696=1195.753,306.154,-69.823,-176.578,7.503,148.430
C00697=1195.757,305.906,-69.793,-176.581,7.500,148.430
C00698=1195.761,305.658,-69.762,-176.583,7.497,148.430
C00699=1195.765,305.410,-69.733,-176.586,7.493,148.430
C00700=1195.770,305.162,-69.702,-176.588,7.491,148.430
C00701=1195.774,304.914,-69.672,-176.590,7.488,148.430
C00702=1195.779,304.666,-69.642,-176.593,7.485,148.430
C00703=1195.783,304.417,-69.612,-176.595,7.483,148.430
C00704=1195.787,304.170,-69.582,-176.598,7.480,148.430
C00705=1195.791,303.920,-69.552,-176.601,7.477,148.430
C00706=1195.795,303.673,-69.521,-176.603,7.474,148.430
C00707=1195.800,303.424,-69.491,-176.606,7.472,148.430
C00708=1195.804,303.177,-69.461,-176.608,7.468,148.430
C00709=1195.808,302.928,-69.432,-176.610,7.465,148.430
C00710=1195.813,302.680,-69.402,-176.613,7.463,148.430
C00711=1195.817,302.432,-69.371,-176.615,7.460,148.430
C00712=1195.821,302.184,-69.342,-176.618,7.457,148.430
C00713=1195.826,301.936,-69.311,-176.620,7.455,148.430
C00714=1195.830,301.688,-69.282,-176.623,7.452,148.430
C00715=1195.834,301.439,-69.252,-176.626,7.449,148.430
C00716=1195.839,301.191,-69.222,-176.628,7.447,148.430
C00717=1195.843,300.943,-69.192,-176.630,7.444,148.430
C00718=1195.847,300.695,-69.163,-176.633,7.441,148.431
C00719=1195.851,300.447,-69.133,-176.636,7.438,148.431
C00720=1195.856,300.199,-69.102,-176.638,7.435,148.431
C00721=1195.860,299.950,-69.073,-176.640,7.432,148.430
C00722=1195.864,299.703,-69.043,-176.643,7.429,148.430
C00723=1195.868,299.454,-69.013,-176.645,7.427,148.430
C00724=1195.873,299.206,-68.983,-176.648,7.424,148.430
C00725=1195.877,298.958,-68.954,-176.650,7.421,148.431
C00726=1195.881,298.710,-68.924,-176.653,7.419,148.431
C00727=1195.885,298.462,-68.894,-176.655,7.416,148.431
C00728=1195.890,298.213,-68.864,-176.658,7.413,148.431
C00729=1195.894,297.965,-68.835,-176.660,7.410,148.431
C00730=1195.898,297.717,-68.805,-176.663,7.407,148.431
C00731=1195.903,297.468,-68.776,-176.666,7.404,148.431
C00732=1195.906,297.221,-68.746,-176.668,7.402,148.431
C00733=1195.911,296.972,-68.716,-176.670,7.399,148.431
C00734=1195.916,296.724,-68.686,-176.673,7.396,148.431
C00735=1195.920,296.476,-68.657,-176.675,7.394,148.431
C00736=1195.924,296.227,-68.627,-176.678,7.391,148.431
C00737=1195.928,295.979,-68.598,-176.681,7.388,148.431
C00738=1195.932,295.731,-68.568,-176.683,7.386,148.431
C00739=1195.937,295.482,-68.539,-176.685,7.383,148.431
C00740=1195.941,295.234,-68.509,-176.688,7.380,148.431
C00741=1195.945,294.986,-68.480,-176.690,7.378,148.431
C00742=1195.950,294.738,-68.450,-176.693,7.375,148.431
C00743=1195.955,294.490,-68.421,-176.696,7.372,148.431
C00744=1195.959,294.242,-68.391,-176.698,7.369,148.431
C00745=1195.963,293.993,-68.362,-176.701,7.366,148.431
C00746=1195.967,293.745,-68.333,-176.703,7.363,148.431
C00747=1195.971,293.497,-68.303,-176.705,7.361,148.431
C00748=1195.975,293.248,-68.274,-176.708,7.358,148.431
C00749=1195.980,293.000,-68.244,-176.711,7.355,148.431
C00750=1195.984,292.752,-68.215,-176.713,7.353,148.431
C00751=1195.989,292.504,-68.186,-176.716,7.350,148.431
C00752=1195.993,292.256,-68.156,-176.718,7.347,148.432
C00753=1195.997,292.008,-68.127,-176.721,7.345,148.432
C00754=1196.001,291.760,-68.097,-176.723,7.342,148.432
C00755=1196.005,291.511,-68.068,-176.726,7.339,148.432
C00756=1196.010,291.262,-68.039,-176.729,7.337,148.432
C00757=1196.014,291.014,-68.010,-176.731,7.334,148.432
C00758=1196.019,290.767,-67.981,-176.733,7.332,148.432
C00759=1196.023,290.518,-67.951,-176.736,7.329,148.432
C00760=1196.027,290.270,-67.922,-176.739,7.326,148.432
C00761=1196.032,290.021,-67.893,-176.741,7.324,148.432
C00762=1196.036,289.773,-67.863,-176.744,7.321,148.432
C00763=1196.040,289.526,-67.835,-176.746,7.318,148.432
C00764=1196.044,289.277,-67.805,-176.748,7.315,148.432
C00765=1196.049,289.002,-67.773,-176.751,7.312,148.432
C00766=1196.054,288.728,-67.741,-176.754,7.309,148.432
C00767=1196.058,288.454,-67.709,-176.757,7.307,148.433
C00768=1196.064,288.179,-67.677,-176.760,7.304,148.433
C00769=1196.068,287.931,-67.647,-176.762,7.301,148.433
C00770=1196.071,287.683,-67.618,-176.765,7.298,148.433
C00771=1196.076,287.434,-67.590,-176.767,7.295,148.433
C00772=1196.081,287.187,-67.561,-176.770,7.292,148.433
C00773=1196.085,286.938,-67.532,-176.772,7.290,148.433
C00774=1196.089,286.689,-67.502,-176.775,7.287,148.433
C00775=1196.094,286.441,-67.473,-176.778,7.285,148.433
C00776=1196.098,286.193,-67.445,-176.780,7.282,148.433
C00777=1196.102,285.945,-67.416,-176.783,7.279,148.433
C00778=1196.107,285.696,-67.387,-176.785,7.277,148.433
C00779=1196.111,285.448,-67.357,-176.788,7.274,148.433
C00780=1196.116,285.200,-67.329,-176.790,7.271,148.433
C00781=1196.119,284.952,-67.300,-176.793,7.269,148.433
C00782=1196.124,284.703,-67.271,-176.795,7.266,148.433
C00783=1196.129,284.455,-67.242,-176.797,7.264,148.433
C00784=1196.133,284.207,-67.213,-176.801,7.261,148.434
C00785=1196.137,283.958,-67.185,-176.803,7.258,148.434
C00786=1196.141,283.709,-67.156,-176.805,7.256,148.434
C00787=1196.146,283.462,-67.127,-176.808,7.253,148.434
C00788=1196.150,283.213,-67.098,-176.810,7.251,148.434
C00789=1196.154,282.965,-67.069,-176.813,7.248,148.434
C00790=1196.159,282.717,-67.041,-176.816,7.245,148.434
C00791=1196.163,282.469,-67.012,-176.818,7.243,148.434
C00792=1196.167,282.220,-66.983,-176.821,7.240,148.434
C00793=1196.172,281.972,-66.955,-176.823,7.238,148.434
C00794=1196.176,281.724,-66.926,-176.826,7.235,148.434
C00795=1196.180,281.475,-66.897,-176.829,7.232,148.434
C00796=1196.185,281.227,-66.869,-176.831,7.229,148.435
C00797=1196.189,280.979,-66.840,-176.834,7.227,148.435
C00798=1196.193,280.731,-66.812,-176.836,7.225,148.435
C00799=1196.198,280.482,-66.783,-176.839,7.222,148.435
C00800=1196.202,280.234,-66.754,-176.841,7.219,148.435
C00801=1196.206,279.986,-66.726,-176.844,7.216,148.435
C00802=1196.211,279.737,-66.697,-176.846,7.213,148.435
C00803=1196.214,279.489,-66.668,-176.849,7.212,148.435
C00804=1196.219,279.241,-66.640,-176.852,7.209,148.435
C00805=1196.224,278.992,-66.611,-176.854,7.206,148.435
C00806=1196.228,278.744,-66.583,-176.857,7.203,148.435
C00807=1196.233,278.495,-66.555,-176.859,7.201,148.436
C00808=1196.236,278.247,-66.526,-176.862,7.199,148.436
C00809=1196.241,277.999,-66.497,-176.865,7.196,148.436
C00810=1196.245,277.750,-66.469,-176.867,7.193,148.436
C00811=1196.250,277.502,-66.441,-176.869,7.190,148.436
C00812=1196.254,277.254,-66.413,-176.872,7.188,148.436
C00813=1196.259,277.005,-66.384,-176.875,7.185,148.436
C00814=1196.262,276.757,-66.356,-176.877,7.183,148.436
C00815=1196.267,276.508,-66.327,-176.880,7.180,148.436
C00816=1196.271,276.261,-66.299,-176.882,7.178,148.436
C00817=1196.276,276.012,-66.270,-176.884,7.175,148.436
C00818=1196.280,275.764,-66.242,-176.888,7.172,148.437
C00819=1196.285,275.515,-66.214,-176.890,7.170,148.437
C00820=1196.289,275.267,-66.186,-176.893,7.167,148.437
C00821=1196.293,275.018,-66.157,-176.895,7.165,148.437
C00822=1196.298,274.770,-66.129,-176.898,7.162,148.437
C00823=1196.302,274.521,-66.101,-176.900,7.160,148.437
C00824=1196.307,274.274,-66.073,-176.903,7.157,148.437
C00825=1196.310,274.025,-66.045,-176.905,7.155,148.437
C00826=1196.315,273.777,-66.016,-176.908,7.152,148.437
C00827=1196.319,273.528,-65.988,-176.910,7.150,148.438
C00828=1196.324,273.280,-65.960,-176.913,7.147,148.438
C00829=1196.328,273.031,-65.932,-176.915,7.145,148.438
C00830=1196.332,272.784,-65.904,-176.918,7.142,148.438
C00831=1196.337,272.535,-65.875,-176.921,7.139,148.438
C00832=1196.341,272.287,-65.847,-176.923,7.137,148.438
C00833=1196.345,272.038,-65.819,-176.926,7.134,148.438
C00834=1196.350,271.789,-65.792,-176.928,7.132,148.438
C00835=1196.354,271.541,-65.764,-176.931,7.129,148.439
C00836=1196.358,271.293,-65.736,-176.933,7.127,148.439
C00837=1196.363,271.044,-65.707,-176.936,7.124,148.439
C00838=1196.367,270.796,-65.679,-176.938,7.122,148.439
C00839=1196.372,270.548,-65.651,-176.941,7.119,148.439
C00840=1196.376,270.299,-65.623,-176.943,7.117,148.439
C00841=1196.381,270.051,-65.596,-176.946,7.114,148.439
C00842=1196.385,269.802,-65.568,-176.949,7.112,148.439
C00843=1196.390,269.554,-65.539,-176.951,7.109,148.439
C00844=1196.393,269.306,-65.511,-176.954,7.107,148.440
C00845=1196.398,269.057,-65.484,-176.956,7.104,148.440
C00846=1196.402,268.809,-65.456,-176.959,7.102,148.440
C00847=1196.407,268.560,-65.427,-176.962,7.099,148.440
C00848=1196.412,268.312,-65.400,-176.964,7.097,148.440
C00849=1196.416,268.064,-65.373,-176.967,7.094,148.440
C00850=1196.420,267.815,-65.344,-176.969,7.092,148.440
C00851=1196.425,267.567,-65.317,-176.972,7.089,148.440
C00852=1196.429,267.318,-65.289,-176.974,7.087,148.441
C00853=1196.433,267.070,-65.261,-176.977,7.084,148.441
C00854=1196.438,266.822,-65.234,-176.979,7.082,148.441
C00855=1196.442,266.573,-65.206,-176.982,7.079,148.441
C00856=1196.446,266.325,-65.178,-176.985,7.077,148.441
C00857=1196.451,266.076,-65.150,-176.987,7.074,148.441
C00858=1196.455,265.828,-65.122,-176.990,7.072,148.441
C00859=1196.460,265.579,-65.095,-176.993,7.069,148.442
C00860=1196.464,265.331,-65.067,-176.995,7.067,148.442
C00861=1196.468,265.082,-65.040,-176.998,7.064,148.442
C00862=1196.472,264.834,-65.012,-177.000,7.062,148.442
C00863=1196.477,264.586,-64.985,-177.002,7.060,148.442
C00864=1196.482,264.337,-64.956,-177.005,7.057,148.442
C00865=1196.486,264.088,-64.929,-177.008,7.055,148.442
C00866=1196.491,263.841,-64.901,-177.010,7.052,148.442
C00867=1196.495,263.591,-64.874,-177.013,7.050,148.443
C00868=1196.499,263.344,-64.846,-177.016,7.048,148.443
C00869=1196.504,263.071,-64.816,-177.018,7.045,148.443
C00870=1196.508,262.798,-64.786,-177.021,7.043,148.443
C00871=1196.513,262.525,-64.756,-177.024,7.040,148.443
C00872=1196.519,262.253,-64.725,-177.027,7.037,148.443
C00873=1196.523,262.003,-64.698,-177.029,7.035,148.444
C00874=1196.527,261.755,-64.671,-177.032,7.032,148.444
C00875=1196.532,261.507,-64.643,-177.034,7.030,148.444
C00876=1196.536,261.259,-64.616,-177.037,7.027,148.444
C00877=1196.540,261.010,-64.588,-177.039,7.025,148.444
C00878=1196.545,260.762,-64.561,-177.043,7.022,148.444
C00879=1196.550,260.513,-64.534,-177.045,7.020,148.444
C00880=1196.554,260.265,-64.507,-177.047,7.017,148.444
C00881=1196.558,260.016,-64.478,-177.050,7.015,148.445
C00882=1196.563,259.767,-64.451,-177.052,7.013,148.445
C00883=1196.567,259.519,-64.424,-177.055,7.010,148.445
C00884=1196.572,259.271,-64.396,-177.058,7.008,148.445
C00885=1196.575,259.023,-64.370,-177.060,7.005,148.445
C00886=1196.580,258.774,-64.343,-177.063,7.003,148.446
C00887=1196.584,258.525,-64.316,-177.066,7.000,148.446
C00888=1196.589,258.277,-64.288,-177.068,6.998,148.446
C00889=1196.593,258.029,-64.261,-177.070,6.996,148.446
C00890=1196.598,257.780,-64.234,-177.073,6.993,148.446
C00891=1196.602,257.531,-64.206,-177.076,6.991,148.446
C00892=1196.607,257.283,-64.179,-177.078,6.988,148.446
C00893=1196.611,257.034,-64.152,-177.081,6.986,148.446
C00894=1196.616,256.786,-64.124,-177.084,6.984,148.447
C00895=1196.620,256.538,-64.098,-177.086,6.981,148.447
C00896=1196.624,256.290,-64.071,-177.089,6.980,148.447
C00897=1196.628,256.040,-64.043,-177.091,6.977,148.447
C00898=1196.633,255.792,-64.016,-177.093,6.974,148.447
C00899=1196.638,255.543,-63.989,-177.097,6.972,148.448
C00900=1196.642,255.295,-63.962,-177.099,6.969,148.448
C00901=1196.646,255.047,-63.936,-177.101,6.968,148.448
C00902=1196.651,254.798,-63.909,-177.104,6.965,148.448
C00903=1196.655,254.550,-63.882,-177.106,6.962,148.448
C00904=1196.659,254.301,-63.854,-177.109,6.960,148.448
C00905=1196.664,254.052,-63.827,-177.112,6.958,148.448
C00906=1196.668,253.804,-63.801,-177.114,6.956,148.449
C00907=1196.673,253.555,-63.774,-177.117,6.953,148.449
C00908=1196.677,253.307,-63.747,-177.120,6.951,148.449
C00909=1196.682,253.058,-63.719,-177.122,6.948,148.449
C00910=1196.686,252.810,-63.693,-177.125,6.946,148.450
C00911=1196.691,252.562,-63.666,-177.127,6.944,148.450
C00912=1196.695,252.313,-63.639,-177.130,6.941,148.450
C00913=1196.700,252.065,-63.612,-177.132,6.939,148.450
C00914=1196.704,251.817,-63.585,-177.135,6.937,148.450
C00915=1196.708,251.567,-63.558,-177.138,6.934,148.450
C00916=1196.713,251.319,-63.531,-177.140,6.932,148.450
C00917=1196.716,251.071,-63.504,-177.143,6.929,148.451
C00918=1196.721,250.822,-63.478,-177.145,6.927,148.451
C00919=1196.726,250.573,-63.451,-177.148,6.925,148.451
C00920=1196.730,250.325,-63.425,-177.151,6.922,148.451
C00921=1196.735,250.076,-63.397,-177.153,6.920,148.451
C00922=1196.739,249.828,-63.370,-177.155,6.918,148.452
C00923=1196.743,249.580,-63.344,-177.158,6.915,148.452
C00924=1196.748,249.331,-63.318,-177.161,6.914,148.452
C00925=1196.753,249.082,-63.291,-177.163,6.911,148.452
C00926=1196.757,248.834,-63.264,-177.166,6.909,148.452
C00927=1196.761,248.585,-63.237,-177.168,6.907,148.452
C00928=1196.766,248.337,-63.211,-177.171,6.904,148.453
C00929=1196.770,248.088,-63.184,-177.174,6.902,148.453
C00930=1196.775,247.840,-63.157,-177.176,6.900,148.453
C00931=1196.779,247.591,-63.131,-177.179,6.897,148.453
C00932=1196.784,247.342,-63.104,-177.182,6.895,148.453
C00933=1196.788,247.094,-63.078,-177.184,6.893,148.454
C00934=1196.793,246.845,-63.051,-177.187,6.890,148.454
C00935=1196.797,246.597,-63.025,-177.189,6.888,148.454
C00936=1196.801,246.348,-62.998,-177.192,6.886,148.454
C00937=1196.806,246.100,-62.972,-177.194,6.883,148.454
C00938=1196.810,245.851,-62.945,-177.197,6.881,148.455
C00939=1196.815,245.603,-62.918,-177.199,6.879,148.455
C00940=1196.819,245.354,-62.892,-177.202,6.877,148.455
C00941=1196.824,245.105,-62.865,-177.205,6.874,148.455
C00942=1196.828,244.856,-62.840,-177.207,6.873,148.455
C00943=1196.832,244.608,-62.813,-177.210,6.870,148.455
C00944=1196.837,244.360,-62.786,-177.213,6.868,148.456
C00945=1196.841,244.112,-62.761,-177.215,6.866,148.456
C00946=1196.846,243.863,-62.734,-177.218,6.863,148.456
C00947=1196.850,243.614,-62.708,-177.220,6.861,148.456
C00948=1196.855,243.366,-62.681,-177.223,6.859,148.457
C00949=1196.859,243.117,-62.655,-177.225,6.856,148.457
C00950=1196.864,242.869,-62.628,-177.228,6.854,148.457
C00951=1196.868,242.620,-62.602,-177.230,6.852,148.457
C00952=1196.872,242.371,-62.576,-177.233,6.849,148.457
C00953=1196.877,242.122,-62.549,-177.236,6.847,148.458
C00954=1196.882,241.874,-62.524,-177.238,6.845,148.458
C00955=1196.886,241.626,-62.497,-177.241,6.843,148.458
C00956=1196.891,241.377,-62.471,-177.244,6.840,148.458
C00957=1196.894,241.129,-62.445,-177.246,6.839,148.458
C00958=1196.899,240.880,-62.418,-177.248,6.836,148.459
C00959=1196.904,240.631,-62.393,-177.252,6.834,148.459
C00960=1196.908,240.382,-62.366,-177.254,6.832,148.459
C00961=1196.913,240.134,-62.340,-177.256,6.830,148.459
C00962=1196.917,239.886,-62.314,-177.259,6.827,148.459
C00963=1196.922,239.637,-62.287,-177.262,6.825,148.460
C00964=1196.926,239.388,-62.262,-177.264,6.823,148.460
C00965=1196.931,239.139,-62.236,-177.267,6.820,148.460
C00966=1196.935,238.891,-62.209,-177.270,6.818,148.460
C00967=1196.940,238.643,-62.183,-177.272,6.816,148.460
C00968=1196.944,238.394,-62.158,-177.275,6.814,148.461
C00969=1196.948,238.145,-62.132,-177.277,6.811,148.461
C00970=1196.953,237.897,-62.105,-177.280,6.809,148.461
C00971=1196.957,237.648,-62.079,-177.283,6.808,148.461
C00972=1196.962,237.399,-62.053,-177.285,6.805,148.461
C00973=1196.967,237.129,-62.025,-177.288,6.803,148.462
C00974=1196.972,236.856,-61.996,-177.291,6.800,148.462
C00975=1196.977,236.584,-61.968,-177.293,6.798,148.462
C00976=1196.982,236.314,-61.940,-177.296,6.795,148.462
C00977=1196.986,236.065,-61.914,-177.299,6.793,148.463
C00978=1196.990,235.816,-61.888,-177.301,6.791,148.463
C00979=1196.995,235.567,-61.862,-177.304,6.789,148.463
C00980=1197.000,235.319,-61.837,-177.307,6.786,148.463
C00981=1197.004,235.070,-61.811,-177.309,6.785,148.464
C00982=1197.008,234.822,-61.784,-177.312,6.783,148.464
C00983=1197.012,234.573,-61.759,-177.315,6.780,148.464
C00984=1197.017,234.325,-61.733,-177.317,6.778,148.464
C00985=1197.022,234.076,-61.707,-177.320,6.776,148.465
C00986=1197.026,233.827,-61.681,-177.322,6.774,148.465
C00987=1197.030,233.578,-61.655,-177.325,6.771,148.465
C00988=1197.035,233.330,-61.630,-177.327,6.769,148.465
C00989=1197.040,233.081,-61.604,-177.330,6.767,148.465
C00990=1197.044,232.833,-61.579,-177.333,6.765,148.466
C00991=1197.049,232.585,-61.553,-177.335,6.762,148.466
C00992=1197.053,232.336,-61.527,-177.338,6.761,148.466
C00993=1197.058,232.087,-61.501,-177.340,6.758,148.466
C00994=1197.063,231.839,-61.476,-177.343,6.757,148.467
C00995=1197.067,231.590,-61.450,-177.346,6.754,148.467
C00996=1197.071,231.341,-61.424,-177.348,6.752,148.467
C00997=1197.076,231.093,-61.399,-177.351,6.750,148.467
C00998=1197.080,230.843,-61.374,-177.353,6.748,148.468
C00999=1197.085,230.595,-61.348,-177.356,6.745,148.468
C01000=1197.089,230.346,-61.323,-177.359,6.743,148.468
C01001=1197.094,230.098,-61.297,-177.361,6.741,148.468
C01002=1197.098,229.849,-61.271,-177.364,6.739,148.468
C01003=1197.103,229.601,-61.246,-177.367,6.737,148.469
C01004=1197.107,229.352,-61.220,-177.369,6.735,148.469
C01005=1197.111,229.103,-61.194,-177.372,6.733,148.469
C01006=1197.116,228.854,-61.170,-177.374,6.731,148.470
C01007=1197.121,228.606,-61.144,-177.378,6.728,148.470
C01008=1197.125,228.357,-61.118,-177.380,6.726,148.470
C01009=1197.130,228.109,-61.093,-177.382,6.724,148.470
C01010=1197.134,227.860,-61.067,-177.385,6.722,148.471
C01011=1197.139,227.611,-61.042,-177.387,6.720,148.471
C01012=1197.143,227.362,-61.017,-177.390,6.718,148.471
C01013=1197.147,227.114,-60.991,-177.393,6.716,148.471
C01014=1197.153,226.865,-60.966,-177.395,6.714,148.471
C01015=1197.157,226.616,-60.940,-177.398,6.712,148.472
C01016=1197.162,226.368,-60.915,-177.401,6.709,148.472
C01017=1197.166,226.119,-60.889,-177.403,6.707,148.472
C01018=1197.170,225.870,-60.865,-177.406,6.705,148.472
C01019=1197.174,225.622,-60.839,-177.408,6.703,148.473
C01020=1197.179,225.373,-60.814,-177.411,6.701,148.473
C01021=1197.184,225.124,-60.789,-177.414,6.698,148.473
C01022=1197.188,224.876,-60.763,-177.416,6.697,148.474
C01023=1197.193,224.628,-60.738,-177.419,6.694,148.474
C01024=1197.197,224.378,-60.713,-177.421,6.693,148.474
C01025=1197.202,224.130,-60.687,-177.424,6.691,148.474
C01026=1197.206,223.881,-60.663,-177.427,6.688,148.475
C01027=1197.210,223.632,-60.637,-177.429,6.686,148.475
C01028=1197.215,223.383,-60.613,-177.432,6.684,148.475
C01029=1197.220,223.135,-60.587,-177.435,6.682,148.475
C01030=1197.224,222.886,-60.561,-177.437,6.680,148.475
C01031=1197.229,222.637,-60.536,-177.440,6.678,148.476
C01032=1197.233,222.389,-60.512,-177.443,6.676,148.476
C01033=1197.238,222.140,-60.487,-177.445,6.674,148.476
C01034=1197.242,221.892,-60.461,-177.447,6.672,148.477
C01035=1197.247,221.642,-60.436,-177.450,6.670,148.477
C01036=1197.251,221.394,-60.411,-177.453,6.668,148.477
C01037=1197.256,221.145,-60.386,-177.455,6.665,148.477
C01038=1197.261,220.896,-60.362,-177.458,6.663,148.478
C01039=1197.265,220.648,-60.336,-177.461,6.661,148.478
C01040=1197.269,220.399,-60.312,-177.463,6.660,148.478
C01041=1197.273,220.150,-60.286,-177.465,6.657,148.478
C01042=1197.279,219.902,-60.261,-177.469,6.655,148.479
C01043=1197.283,219.653,-60.236,-177.471,6.653,148.479
C01044=1197.287,219.404,-60.212,-177.474,6.651,148.479
C01045=1197.292,219.156,-60.187,-177.476,6.649,148.479
C01046=1197.297,218.907,-60.161,-177.479,6.647,148.480
C01047=1197.301,218.658,-60.137,-177.481,6.645,148.480
C01048=1197.306,218.409,-60.112,-177.485,6.643,148.480
C01049=1197.310,218.161,-60.087,-177.487,6.641,148.481
C01050=1197.314,217.912,-60.062,-177.489,6.639,148.481
C01051=1197.319,217.663,-60.038,-177.492,6.637,148.481
C01052=1197.324,217.415,-60.012,-177.495,6.635,148.482
C01053=1197.328,217.166,-59.988,-177.497,6.633,148.482
C01054=1197.333,216.917,-59.963,-177.500,6.630,148.482
C01055=1197.337,216.668,-59.939,-177.503,6.628,148.482
C01056=1197.342,216.420,-59.913,-177.505,6.627,148.483
C01057=1197.347,216.171,-59.889,-177.508,6.625,148.483
C01058=1197.351,215.922,-59.864,-177.510,6.623,148.483
C01059=1197.356,215.673,-59.839,-177.513,6.621,148.483
C01060=1197.359,215.424,-59.815,-177.516,6.618,148.484
C01061=1197.364,215.176,-59.790,-177.519,6.616,148.484
C01062=1197.369,214.927,-59.765,-177.521,6.614,148.484
C01063=1197.373,214.678,-59.740,-177.524,6.612,148.484
C01064=1197.378,214.430,-59.716,-177.526,6.611,148.485
C01065=1197.383,214.181,-59.692,-177.529,6.609,148.485
C01066=1197.387,213.932,-59.667,-177.532,6.607,148.485
C01067=1197.391,213.684,-59.642,-177.534,6.604,148.486
C01068=1197.397,213.435,-59.617,-177.537,6.602,148.486
C01069=1197.400,213.186,-59.593,-177.540,6.600,148.486
C01070=1197.405,212.937,-59.568,-177.542,6.598,148.487
C01071=1197.410,212.689,-59.544,-177.545,6.597,148.487
C01072=1197.414,212.440,-59.519,-177.547,6.594,148.487
C01073=1197.419,212.191,-59.495,-177.550,6.593,148.487
C01074=1197.424,211.942,-59.470,-177.553,6.590,148.488
C01075=1197.428,211.693,-59.446,-177.556,6.588,148.488
C01076=1197.433,211.445,-59.421,-177.558,6.586,148.488
C01077=1197.438,211.174,-59.394,-177.561,6.585,148.489
C01078=1197.442,210.905,-59.368,-177.564,6.582,148.489
C01079=1197.447,210.633,-59.342,-177.567,6.580,148.489
C01080=1197.452,210.363,-59.315,-177.569,6.578,148.490
C01081=1197.457,210.114,-59.291,-177.572,6.575,148.490
C01082=1197.461,209.865,-59.266,-177.575,6.573,148.490
C01083=1197.466,209.617,-59.242,-177.577,6.572,148.490
C01084=1197.471,209.368,-59.217,-177.580,6.570,148.491
C01085=1197.475,209.119,-59.193,-177.583,6.568,148.491
C01086=1197.479,208.870,-59.169,-177.585,6.566,148.491
C01087=1197.484,208.622,-59.144,-177.587,6.564,148.492
C01088=1197.489,208.373,-59.120,-177.590,6.562,148.492
C01089=1197.494,208.124,-59.096,-177.593,6.560,148.492
C01090=1197.498,207.875,-59.072,-177.596,6.558,148.493
C01091=1197.502,207.626,-59.048,-177.599,6.556,148.493
C01092=1197.507,207.378,-59.023,-177.601,6.554,148.493
C01093=1197.512,207.129,-58.999,-177.603,6.552,148.493
C01094=1197.516,206.881,-58.975,-177.606,6.550,148.494
C01095=1197.521,206.631,-58.951,-177.609,6.548,148.494
C01096=1197.525,206.382,-58.926,-177.611,6.546,148.494
C01097=1197.530,206.134,-58.902,-177.614,6.545,148.495
C01098=1197.535,205.885,-58.878,-177.617,6.543,148.495
C01099=1197.540,205.636,-58.854,-177.619,6.541,148.495
C01100=1197.543,205.387,-58.830,-177.622,6.538,148.495
C01101=1197.548,205.139,-58.806,-177.625,6.536,148.496
C01102=1197.553,204.890,-58.781,-177.627,6.534,148.496
C01103=1197.558,204.641,-58.758,-177.630,6.533,148.496
C01104=1197.562,204.392,-58.734,-177.633,6.531,148.497
C01105=1197.566,204.144,-58.710,-177.635,6.529,148.497
C01106=1197.571,203.894,-58.685,-177.638,6.527,148.497
C01107=1197.576,203.646,-58.661,-177.640,6.525,148.498
C01108=1197.580,203.397,-58.637,-177.643,6.523,148.498
C01109=1197.585,203.148,-58.614,-177.646,6.521,148.498
C01110=1197.589,202.900,-58.590,-177.648,6.520,148.499
C01111=1197.594,202.651,-58.565,-177.651,6.518,148.499
C01112=1197.598,202.401,-58.541,-177.653,6.516,148.499
C01113=1197.603,202.153,-58.517,-177.656,6.513,148.499
C01114=1197.607,201.904,-58.494,-177.659,6.511,148.500
C01115=1197.612,201.655,-58.470,-177.662,6.509,148.500
C01116=1197.616,201.406,-58.447,-177.664,6.508,148.500
C01117=1197.622,201.158,-58.422,-177.667,6.506,148.501
C01118=1197.626,200.909,-58.398,-177.669,6.504,148.501
C01119=1197.631,200.660,-58.374,-177.672,6.502,148.501
C01120=1197.635,200.412,-58.350,-177.675,6.500,148.502
C01121=1197.639,200.162,-58.327,-177.677,6.498,148.502
C01122=1197.644,199.914,-58.303,-177.680,6.496,148.502
C01123=1197.648,199.665,-58.279,-177.682,6.494,148.503
C01124=1197.653,199.416,-58.255,-177.685,6.493,148.503
C01125=1197.657,199.167,-58.232,-177.688,6.491,148.503
C01126=1197.663,198.918,-58.208,-177.690,6.489,148.504
C01127=1197.667,198.669,-58.184,-177.693,6.487,148.504
C01128=1197.672,198.420,-58.160,-177.696,6.485,148.504
C01129=1197.676,198.172,-58.136,-177.698,6.484,148.505
C01130=1197.681,197.923,-58.113,-177.701,6.482,148.505
C01131=1197.685,197.675,-58.089,-177.703,6.480,148.505
C01132=1197.690,197.426,-58.066,-177.706,6.477,148.505
C01133=1197.695,197.176,-58.042,-177.709,6.475,148.506
C01134=1197.699,196.928,-58.018,-177.712,6.473,148.506
C01135=1197.704,196.679,-57.995,-177.714,6.472,148.507
C01136=1197.709,196.430,-57.971,-177.717,6.470,148.507
C01137=1197.713,196.182,-57.947,-177.720,6.468,148.507
C01138=1197.718,195.933,-57.924,-177.722,6.466,148.508
C01139=1197.722,195.684,-57.901,-177.725,6.464,148.508
C01140=1197.727,195.435,-57.876,-177.728,6.463,148.508
C01141=1197.731,195.186,-57.853,-177.730,6.461,148.509
C01142=1197.736,194.937,-57.830,-177.733,6.459,148.509
C01143=1197.741,194.688,-57.806,-177.735,6.457,148.509
C01144=1197.745,194.440,-57.782,-177.738,6.455,148.509
C01145=1197.750,194.191,-57.759,-177.740,6.453,148.510
C01146=1197.755,193.942,-57.736,-177.743,6.451,148.510
C01147=1197.759,193.693,-57.712,-177.746,6.449,148.510
C01148=1197.763,193.444,-57.690,-177.748,6.448,148.511
C01149=1197.768,193.195,-57.665,-177.751,6.446,148.511
C01150=1197.772,192.946,-57.642,-177.754,6.444,148.512
C01151=1197.777,192.697,-57.619,-177.756,6.442,148.512
C01152=1197.782,192.448,-57.595,-177.759,6.440,148.512
C01153=1197.787,192.199,-57.572,-177.762,6.439,148.513
C01154=1197.791,191.950,-57.549,-177.764,6.437,148.513
C01155=1197.796,191.702,-57.525,-177.767,6.435,148.513
C01156=1197.800,191.453,-57.501,-177.770,6.433,148.514
C01157=1197.804,191.204,-57.478,-177.772,6.431,148.514
C01158=1197.809,190.955,-57.455,-177.775,6.430,148.514
C01159=1197.814,190.707,-57.432,-177.778,6.428,148.515
C01160=1197.819,190.458,-57.409,-177.780,6.426,148.515
C01161=1197.824,190.209,-57.385,-177.782,6.424,148.515
C01162=1197.828,189.960,-57.362,-177.785,6.422,148.516
C01163=1197.832,189.711,-57.339,-177.788,6.420,148.516
C01164=1197.837,189.462,-57.316,-177.790,6.418,148.516
C01165=1197.842,189.213,-57.293,-177.793,6.417,148.517
C01166=1197.846,188.964,-57.269,-177.796,6.415,148.517
C01167=1197.851,188.715,-57.246,-177.798,6.413,148.517
C01168=1197.856,188.467,-57.223,-177.801,6.411,148.518
C01169=1197.860,188.218,-57.200,-177.804,6.409,148.518
C01170=1197.865,187.969,-57.177,-177.806,6.408,148.518
C01171=1197.870,187.720,-57.153,-177.809,6.406,148.519
C01172=1197.874,187.471,-57.131,-177.812,6.404,148.519
C01173=1197.878,187.222,-57.107,-177.814,6.403,148.519
C01174=1197.883,186.973,-57.084,-177.816,6.401,148.520
C01175=1197.888,186.725,-57.061,-177.819,6.399,148.520
C01176=1197.892,186.476,-57.038,-177.822,6.398,148.520
C01177=1197.897,186.227,-57.015,-177.824,6.396,148.521
C01178=1197.902,185.977,-56.992,-177.827,6.394,148.521
C01179=1197.906,185.728,-56.969,-177.830,6.392,148.522
C01180=1197.911,185.479,-56.946,-177.832,6.390,148.522
C01181=1197.916,185.210,-56.921,-177.835,6.389,148.522
C01182=1197.921,184.940,-56.896,-177.838,6.386,148.523
C01183=1197.926,184.670,-56.871,-177.841,6.384,148.523
C01184=1197.931,184.401,-56.846,-177.844,6.383,148.524
C01185=1197.936,184.153,-56.824,-177.847,6.381,148.524
C01186=1197.941,183.904,-56.801,-177.849,6.379,148.524
C01187=1197.945,183.655,-56.778,-177.852,6.377,148.525
C01188=1197.949,183.406,-56.755,-177.855,6.375,148.525
C01189=1197.954,183.156,-56.732,-177.857,6.374,148.525
C01190=1197.959,182.908,-56.710,-177.860,6.372,148.526
C01191=1197.964,182.659,-56.686,-177.863,6.370,148.526
C01192=1197.968,182.410,-56.663,-177.865,6.369,148.526
C01193=1197.973,182.161,-56.641,-177.867,6.367,148.527
C01194=1197.978,181.912,-56.618,-177.870,6.365,148.527
C01195=1197.982,181.664,-56.595,-177.873,6.364,148.527
C01196=1197.987,181.414,-56.572,-177.875,6.362,148.528
C01197=1197.991,181.165,-56.550,-177.878,6.360,148.528
C01198=1197.996,180.917,-56.527,-177.881,6.358,148.529
C01199=1198.000,180.668,-56.505,-177.883,6.356,148.529
C01200=1198.005,180.419,-56.481,-177.886,6.355,148.529
C01201=1198.009,180.170,-56.458,-177.889,6.353,148.530
C01202=1198.015,179.921,-56.436,-177.891,6.351,148.530
C01203=1198.019,179.672,-56.413,-177.894,6.349,148.530
C01204=1198.024,179.423,-56.391,-177.897,6.347,148.531
C01205=1198.028,179.175,-56.368,-177.899,6.346,148.531
C01206=1198.033,178.925,-56.346,-177.902,6.345,148.531
C01207=1198.037,178.676,-56.323,-177.904,6.343,148.532
C01208=1198.042,178.428,-56.300,-177.907,6.341,148.532
C01209=1198.047,178.178,-56.278,-177.910,6.339,148.532
C01210=1198.051,177.929,-56.255,-177.912,6.337,148.533
C01211=1198.056,177.681,-56.233,-177.915,6.336,148.533
C01212=1198.061,177.432,-56.209,-177.918,6.334,148.534
C01213=1198.065,177.182,-56.187,-177.920,6.332,148.534
C01214=1198.070,176.934,-56.164,-177.923,6.330,148.534
C01215=1198.075,176.685,-56.142,-177.925,6.329,148.535
C01216=1198.079,176.436,-56.120,-177.928,6.327,148.535
C01217=1198.084,176.187,-56.097,-177.930,6.326,148.535
C01218=1198.089,175.938,-56.075,-177.933,6.324,148.536
C01219=1198.093,175.689,-56.052,-177.936,6.322,148.536
C01220=1198.098,175.440,-56.030,-177.939,6.321,148.537
C01221=1198.102,175.191,-56.007,-177.941,6.319,148.537
C01222=1198.107,174.942,-55.985,-177.944,6.317,148.537
C01223=1198.112,174.693,-55.963,-177.947,6.315,148.538
C01224=1198.116,174.444,-55.940,-177.949,6.314,148.538
C01225=1198.122,174.195,-55.918,-177.952,6.312,148.539
C01226=1198.126,173.946,-55.896,-177.954,6.311,148.539
C01227=1198.130,173.697,-55.873,-177.957,6.309,148.539
C01228=1198.135,173.448,-55.851,-177.960,6.307,148.540
C01229=1198.140,173.199,-55.829,-177.962,6.305,148.540
C01230=1198.144,172.951,-55.807,-177.965,6.303,148.540
C01231=1198.149,172.701,-55.784,-177.968,6.302,148.541
C01232=1198.154,172.452,-55.762,-177.970,6.301,148.541
C01233=1198.158,172.204,-55.740,-177.972,6.299,148.541
C01234=1198.163,171.954,-55.717,-177.975,6.297,148.542
C01235=1198.168,171.706,-55.695,-177.978,6.296,148.542
C01236=1198.172,171.456,-55.673,-177.981,6.294,148.543
C01237=1198.177,171.208,-55.651,-177.983,6.292,148.543
C01238=1198.182,170.959,-55.628,-177.986,6.290,148.543
C01239=1198.187,170.710,-55.606,-177.988,6.289,148.544
C01240=1198.191,170.461,-55.584,-177.991,6.287,148.544
C01241=1198.195,170.211,-55.562,-177.994,6.286,148.545
C01242=1198.200,169.963,-55.539,-177.996,6.284,148.545
C01243=1198.205,169.714,-55.517,-177.999,6.282,148.545
C01244=1198.210,169.465,-55.496,-178.002,6.280,148.546
C01245=1198.214,169.216,-55.474,-178.005,6.279,148.546
C01246=1198.220,168.967,-55.451,-178.007,6.278,148.547
C01247=1198.224,168.717,-55.429,-178.010,6.276,148.547
C01248=1198.229,168.469,-55.408,-178.012,6.274,148.547
C01249=1198.233,168.220,-55.385,-178.015,6.272,148.548
C01250=1198.237,167.971,-55.363,-178.018,6.271,148.548
C01251=1198.242,167.722,-55.341,-178.020,6.269,148.548
C01252=1198.247,167.473,-55.319,-178.022,6.268,148.549
C01253=1198.252,167.224,-55.297,-178.025,6.266,148.549
C01254=1198.256,166.975,-55.275,-178.028,6.264,148.550
C01255=1198.261,166.726,-55.253,-178.031,6.263,148.550
C01256=1198.266,166.477,-55.231,-178.033,6.261,148.551
C01257=1198.270,166.228,-55.209,-178.036,6.259,148.551
C01258=1198.275,165.979,-55.188,-178.038,6.258,148.551
C01259=1198.280,165.730,-55.165,-178.041,6.257,148.552
C01260=1198.285,165.481,-55.143,-178.044,6.255,148.552
C01261=1198.290,165.232,-55.122,-178.046,6.253,148.552
C01262=1198.294,164.983,-55.100,-178.049,6.251,148.553
C01263=1198.299,164.734,-55.078,-178.052,6.251,148.553
C01264=1198.303,164.485,-55.056,-178.054,6.249,148.554
C01265=1198.308,164.236,-55.034,-178.057,6.247,148.554
C01266=1198.312,163.987,-55.012,-178.060,6.245,148.555
C01267=1198.317,163.738,-54.990,-178.062,6.243,148.555
C01268=1198.322,163.490,-54.969,-178.064,6.242,148.555
C01269=1198.326,163.240,-54.947,-178.067,6.241,148.556
C01270=1198.331,162.991,-54.926,-178.070,6.239,148.556
C01271=1198.335,162.742,-54.904,-178.073,6.237,148.557
C01272=1198.340,162.493,-54.882,-178.075,6.236,148.557
C01273=1198.345,162.244,-54.860,-178.078,6.235,148.557
C01274=1198.350,161.995,-54.838,-178.080,6.233,148.558
C01275=1198.354,161.746,-54.817,-178.083,6.231,148.558
C01276=1198.359,161.497,-54.795,-178.086,6.229,148.558
C01277=1198.364,161.248,-54.774,-178.089,6.228,148.559
C01278=1198.369,160.999,-54.752,-178.091,6.227,148.559
C01279=1198.373,160.750,-54.730,-178.094,6.225,148.560
C01280=1198.378,160.501,-54.708,-178.096,6.223,148.560
C01281=1198.383,160.252,-54.687,-178.099,6.221,148.561
C01282=1198.387,160.003,-54.665,-178.102,6.220,148.561
C01283=1198.392,159.754,-54.643,-178.104,6.219,148.561
C01284=1198.397,159.505,-54.622,-178.107,6.217,148.562
C01285=1198.402,159.236,-54.599,-178.110,6.215,148.562
C01286=1198.407,158.967,-54.576,-178.112,6.214,148.563
C01287=1198.412,158.698,-54.553,-178.115,6.212,148.563
C01288=1198.417,158.429,-54.529,-178.118,6.210,148.564
C01289=1198.422,158.179,-54.507,-178.121,6.209,148.564
C01290=1198.427,157.931,-54.486,-178.123,6.207,148.564
C01291=1198.431,157.682,-54.464,-178.126,6.206,148.565
C01292=1198.435,157.432,-54.443,-178.129,6.204,148.565
C01293=1198.440,157.184,-54.422,-178.131,6.203,148.566
C01294=1198.445,156.935,-54.400,-178.134,6.201,148.566
C01295=1198.450,156.686,-54.379,-178.137,6.199,148.566
C01296=1198.454,156.436,-54.357,-178.139,6.198,148.567
C01297=1198.460,156.187,-54.336,-178.142,6.197,148.567
C01298=1198.464,155.939,-54.315,-178.145,6.195,148.568
C01299=1198.468,155.689,-54.293,-178.147,6.193,148.568
C01300=1198.473,155.440,-54.272,-178.149,6.192,148.569
C01301=1198.478,155.192,-54.250,-178.152,6.190,148.569
C01302=1198.483,154.942,-54.229,-178.155,6.189,148.570
C01303=1198.488,154.693,-54.207,-178.158,6.187,148.570
C01304=1198.492,154.444,-54.187,-178.160,6.186,148.570
C01305=1198.497,154.195,-54.165,-178.163,6.184,148.571
C01306=1198.502,153.946,-54.144,-178.165,6.183,148.571
C01307=1198.506,153.697,-54.122,-178.169,6.181,148.572
C01308=1198.511,153.448,-54.102,-178.171,6.180,148.572
C01309=1198.516,153.199,-54.080,-178.173,6.178,148.572
C01310=1198.521,152.950,-54.059,-178.176,6.177,148.573
C01311=1198.526,152.701,-54.037,-178.178,6.176,148.573
C01312=1198.529,152.452,-54.017,-178.181,6.174,148.574
C01313=1198.535,152.202,-53.996,-178.184,6.172,148.574
C01314=1198.540,151.954,-53.974,-178.187,6.171,148.575
C01315=1198.545,151.704,-53.953,-178.189,6.170,148.575
C01316=1198.549,151.456,-53.932,-178.191,6.168,148.575
C01317=1198.553,151.206,-53.911,-178.195,6.166,148.576
C01318=1198.559,150.957,-53.890,-178.197,6.165,148.576
C01319=1198.563,150.709,-53.869,-178.199,6.164,148.577
C01320=1198.568,150.459,-53.848,-178.202,6.162,148.577
C01321=1198.573,150.211,-53.826,-178.205,6.160,148.577
C01322=1198.577,149.961,-53.805,-178.207,6.160,148.578
C01323=1198.582,149.712,-53.784,-178.210,6.158,148.578
C01324=1198.587,149.463,-53.763,-178.213,6.156,148.579
C01325=1198.591,149.214,-53.742,-178.215,6.154,148.579
C01326=1198.596,148.965,-53.721,-178.218,6.154,148.580
C01327=1198.601,148.716,-53.701,-178.221,6.152,148.580
C01328=1198.605,148.467,-53.679,-178.223,6.150,148.581
C01329=1198.610,148.217,-53.658,-178.225,6.149,148.581
C01330=1198.615,147.968,-53.637,-178.229,6.148,148.582
C01331=1198.620,147.719,-53.616,-178.231,6.146,148.582
C01332=1198.624,147.471,-53.595,-178.234,6.144,148.582
C01333=1198.629,147.222,-53.574,-178.236,6.143,148.583
C01334=1198.634,146.972,-53.553,-178.239,6.141,148.583
C01335=1198.639,146.723,-53.533,-178.242,6.140,148.584
C01336=1198.643,146.473,-53.512,-178.244,6.139,148.584
C01337=1198.647,146.225,-53.491,-178.247,6.137,148.585
C01338=1198.653,145.976,-53.470,-178.249,6.135,148.585
C01339=1198.657,145.727,-53.449,-178.252,6.135,148.586
C01340=1198.662,145.478,-53.428,-178.255,6.133,148.586
C01341=1198.667,145.229,-53.408,-178.257,6.131,148.586
C01342=1198.672,144.979,-53.387,-178.259,6.130,148.587
C01343=1198.676,144.731,-53.366,-178.263,6.129,148.587
C01344=1198.681,144.482,-53.345,-178.265,6.127,148.588
C01345=1198.686,144.233,-53.325,-178.267,6.126,148.588
C01346=1198.691,143.984,-53.304,-178.270,6.124,148.588
C01347=1198.695,143.735,-53.283,-178.273,6.123,148.589
C01348=1198.700,143.485,-53.262,-178.275,6.122,148.589
C01349=1198.704,143.236,-53.242,-178.278,6.120,148.590
C01350=1198.709,142.987,-53.221,-178.281,6.119,148.590
C01351=1198.714,142.738,-53.200,-178.283,6.118,148.591
C01352=1198.719,142.488,-53.179,-178.286,6.116,148.591
C01353=1198.723,142.239,-53.159,-178.289,6.114,148.592
C01354=1198.729,141.990,-53.138,-178.291,6.114,148.592
C01355=1198.733,141.741,-53.118,-178.294,6.112,148.593
C01356=1198.737,141.492,-53.097,-178.297,6.110,148.593
C01357=1198.743,141.243,-53.076,-178.299,6.109,148.593
C01358=1198.747,140.994,-53.056,-178.302,6.108,148.594
C01359=1198.752,140.745,-53.035,-178.305,6.106,148.594
C01360=1198.757,140.496,-53.014,-178.307,6.105,148.595
C01361=1198.761,140.247,-52.994,-178.310,6.103,148.595
C01362=1198.766,139.998,-52.973,-178.313,6.102,148.596
C01363=1198.771,139.749,-52.953,-178.315,6.101,148.596
C01364=1198.776,139.499,-52.932,-178.317,6.099,148.597
C01365=1198.780,139.250,-52.911,-178.321,6.098,148.597
C01366=1198.785,139.001,-52.892,-178.323,6.097,148.598
C01367=1198.790,138.752,-52.871,-178.325,6.095,148.598
C01368=1198.795,138.503,-52.850,-178.329,6.093,148.599
C01369=1198.799,138.254,-52.830,-178.331,6.092,148.599
C01370=1198.804,138.004,-52.809,-178.333,6.091,148.599
C01371=1198.809,137.755,-52.789,-178.336,6.089,148.600
C01372=1198.813,137.507,-52.768,-178.339,6.088,148.600
C01373=1198.818,137.257,-52.749,-178.341,6.087,148.601
C01374=1198.823,137.008,-52.728,-178.343,6.086,148.601
C01375=1198.828,136.759,-52.708,-178.347,6.084,148.602
C01376=1198.833,136.511,-52.687,-178.349,6.082,148.602
C01377=1198.838,136.261,-52.666,-178.351,6.081,148.603
C01378=1198.842,136.012,-52.647,-178.355,6.080,148.603
C01379=1198.847,135.763,-52.626,-178.357,6.078,148.604
C01380=1198.851,135.514,-52.606,-178.359,6.077,148.604
C01381=1198.856,135.265,-52.585,-178.363,6.076,148.605
C01382=1198.861,135.015,-52.565,-178.365,6.075,148.605
C01383=1198.866,134.766,-52.545,-178.367,6.073,148.605
C01384=1198.870,134.517,-52.525,-178.370,6.071,148.606
C01385=1198.876,134.267,-52.504,-178.373,6.071,148.606
C01386=1198.881,134.019,-52.484,-178.375,6.069,148.607
C01387=1198.885,133.770,-52.464,-178.378,6.067,148.607
C01388=1198.890,133.520,-52.444,-178.381,6.067,148.608
C01389=1198.895,133.252,-52.422,-178.383,6.065,148.608
C01390=1198.900,132.983,-52.401,-178.387,6.063,148.609
C01391=1198.905,132.714,-52.378,-178.389,6.062,148.609
C01392=1198.910,132.446,-52.357,-178.392,6.061,148.610
C01393=1198.916,132.197,-52.336,-178.394,6.059,148.610
C01394=1198.920,131.948,-52.317,-178.397,6.057,148.611
C01395=1198.925,131.699,-52.296,-178.400,6.057,148.611
C01396=1198.929,131.449,-52.277,-178.402,6.055,148.612
C01397=1198.934,131.200,-52.256,-178.405,6.054,148.612
C01398=1198.938,130.951,-52.236,-178.408,6.053,148.613
C01399=1198.943,130.702,-52.216,-178.410,6.051,148.613
C01400=1198.949,130.453,-52.196,-178.413,6.050,148.613
C01401=1198.954,130.203,-52.176,-178.416,6.049,148.614
C01402=1198.958,129.955,-52.156,-178.418,6.048,148.614
C01403=1198.963,129.705,-52.136,-178.421,6.046,148.615
C01404=1198.967,129.456,-52.116,-178.423,6.045,148.615
C01405=1198.973,129.207,-52.096,-178.426,6.044,148.616
C01406=1198.977,128.958,-52.076,-178.429,6.042,148.616
C01407=1198.982,128.709,-52.056,-178.431,6.041,148.617
C01408=1198.986,128.460,-52.036,-178.434,6.039,148.617
C01409=1198.991,128.210,-52.016,-178.436,6.039,148.618
C01410=1198.996,127.962,-51.996,-178.439,6.037,148.618
C01411=1199.001,127.712,-51.977,-178.442,6.035,148.619
C01412=1199.005,127.463,-51.957,-178.444,6.035,148.619
C01413=1199.010,127.214,-51.937,-178.447,6.033,148.620
C01414=1199.015,126.965,-51.917,-178.449,6.032,148.620
C01415=1199.020,126.716,-51.897,-178.452,6.031,148.621
C01416=1199.024,126.466,-51.877,-178.455,6.030,148.621
C01417=1199.029,126.217,-51.858,-178.458,6.028,148.622
C01418=1199.034,125.968,-51.837,-178.460,6.027,148.622
C01419=1199.039,125.719,-51.818,-178.463,6.025,148.623
C01420=1199.044,125.469,-51.798,-178.466,6.024,148.623
C01421=1199.048,125.220,-51.778,-178.468,6.023,148.624
C01422=1199.053,124.972,-51.759,-178.471,6.021,148.624
C01423=1199.058,124.722,-51.739,-178.473,6.021,148.625
C01424=1199.063,124.473,-51.719,-178.476,6.019,148.625
C01425=1199.067,124.224,-51.699,-178.478,6.018,148.626
C01426=1199.073,123.975,-51.680,-178.481,6.017,148.626
C01427=1199.077,123.725,-51.660,-178.483,6.016,148.626
C01428=1199.082,123.476,-51.640,-178.486,6.014,148.627
C01429=1199.087,123.227,-51.620,-178.489,6.012,148.627
C01430=1199.092,122.978,-51.601,-178.491,6.012,148.628
C01431=1199.097,122.728,-51.581,-178.494,6.010,148.628
C01432=1199.101,122.479,-51.561,-178.497,6.009,148.629
C01433=1199.106,122.231,-51.542,-178.500,6.008,148.630
C01434=1199.110,121.981,-51.522,-178.502,6.007,148.630
C01435=1199.115,121.732,-51.503,-178.505,6.005,148.630
C01436=1199.121,121.483,-51.483,-178.507,6.004,148.631
C01437=1199.125,121.234,-51.463,-178.510,6.003,148.631
C01438=1199.130,120.984,-51.443,-178.512,6.002,148.632
C01439=1199.135,120.735,-51.424,-178.515,6.000,148.632
C01440=1199.140,120.486,-51.404,-178.517,5.999,148.633
C01441=1199.144,120.236,-51.385,-178.520,5.998,148.633
C01442=1199.149,119.988,-51.366,-178.523,5.997,148.634
C01443=1199.154,119.738,-51.346,-178.526,5.996,148.634
C01444=1199.158,119.489,-51.326,-178.528,5.994,148.635
C01445=1199.164,119.240,-51.307,-178.531,5.993,148.635
C01446=1199.168,118.991,-51.288,-178.534,5.992,148.636
C01447=1199.173,118.742,-51.268,-178.536,5.991,148.636
C01448=1199.178,118.492,-51.249,-178.539,5.989,148.637
C01449=1199.183,118.243,-51.229,-178.541,5.988,148.637
C01450=1199.188,117.994,-51.210,-178.544,5.986,148.638
C01451=1199.192,117.745,-51.191,-178.546,5.986,148.638
C01452=1199.197,117.496,-51.171,-178.549,5.984,148.639
C01453=1199.202,117.246,-51.152,-178.552,5.984,148.639
C01454=1199.207,116.997,-51.132,-178.554,5.982,148.640
C01455=1199.211,116.748,-51.113,-178.557,5.981,148.640
C01456=1199.216,116.499,-51.094,-178.560,5.979,148.641
C01457=1199.221,116.250,-51.074,-178.562,5.978,148.641
C01458=1199.226,116.000,-51.055,-178.565,5.977,148.642
C01459=1199.230,115.751,-51.036,-178.567,5.976,148.642
C01460=1199.236,115.502,-51.016,-178.570,5.975,148.643
C01461=1199.240,115.253,-50.997,-178.573,5.974,148.643
C01462=1199.245,115.004,-50.978,-178.575,5.972,148.644
C01463=1199.250,114.754,-50.958,-178.578,5.971,148.644
C01464=1199.255,114.506,-50.939,-178.581,5.970,148.645
C01465=1199.259,114.256,-50.921,-178.583,5.969,148.645
C01466=1199.265,114.007,-50.902,-178.586,5.967,148.646
C01467=1199.269,113.757,-50.882,-178.588,5.967,148.646
C01468=1199.275,113.508,-50.863,-178.591,5.965,148.647
C01469=1199.279,113.259,-50.844,-178.593,5.964,148.647
C01470=1199.283,113.010,-50.824,-178.596,5.963,148.648
C01471=1199.288,112.761,-50.805,-178.599,5.962,148.648
C01472=1199.293,112.511,-50.786,-178.601,5.961,148.649
C01473=1199.298,112.262,-50.767,-178.604,5.959,148.649
C01474=1199.302,112.013,-50.748,-178.606,5.959,148.650
C01475=1199.308,111.764,-50.729,-178.609,5.957,148.650
C01476=1199.313,111.514,-50.709,-178.612,5.956,148.651
C01477=1199.317,111.265,-50.691,-178.614,5.955,148.651
C01478=1199.322,111.015,-50.671,-178.617,5.954,148.652
C01479=1199.327,110.767,-50.653,-178.620,5.952,148.652
C01480=1199.332,110.517,-50.633,-178.622,5.951,148.653
C01481=1199.336,110.268,-50.615,-178.625,5.950,148.654
C01482=1199.342,110.019,-50.596,-178.627,5.949,148.654
C01483=1199.347,109.770,-50.576,-178.630,5.948,148.655
C01484=1199.351,109.521,-50.557,-178.633,5.947,148.655
C01485=1199.356,109.271,-50.538,-178.636,5.945,148.656
C01486=1199.361,109.022,-50.520,-178.638,5.944,148.656
C01487=1199.366,108.773,-50.500,-178.640,5.944,148.657
C01488=1199.370,108.524,-50.482,-178.643,5.942,148.657
C01489=1199.375,108.274,-50.462,-178.646,5.941,148.658
C01490=1199.380,108.026,-50.444,-178.648,5.940,148.658
C01491=1199.385,107.775,-50.425,-178.651,5.939,148.659
C01492=1199.389,107.527,-50.406,-178.654,5.937,148.659
C01493=1199.395,107.259,-50.385,-178.656,5.937,148.660
C01494=1199.400,106.990,-50.365,-178.659,5.935,148.660
C01495=1199.405,106.722,-50.345,-178.662,5.934,148.661
C01496=1199.410,106.453,-50.324,-178.665,5.933,148.661
C01497=1199.415,106.204,-50.306,-178.668,5.931,148.662
C01498=1199.420,105.955,-50.287,-178.670,5.931,148.663
C01499=1199.424,105.705,-50.268,-178.673,5.929,148.663
C01500=1199.430,105.456,-50.250,-178.675,5.928,148.663
C01501=1199.434,105.207,-50.231,-178.678,5.927,148.664
C01502=1199.440,104.957,-50.212,-178.680,5.926,148.664
C01503=1199.444,104.709,-50.193,-178.683,5.925,148.665
C01504=1199.449,104.459,-50.175,-178.686,5.923,148.665
C01505=1199.454,104.210,-50.156,-178.688,5.923,148.666
C01506=1199.459,103.961,-50.138,-178.691,5.921,148.666
C01507=1199.464,103.711,-50.118,-178.694,5.920,148.667
C01508=1199.469,103.462,-50.100,-178.696,5.920,148.668
C01509=1199.473,103.213,-50.081,-178.699,5.918,148.668
C01510=1199.478,102.963,-50.062,-178.701,5.917,148.669
C01511=1199.483,102.715,-50.044,-178.704,5.916,148.669
C01512=1199.488,102.464,-50.025,-178.706,5.915,148.670
C01513=1199.492,102.216,-50.006,-178.709,5.914,148.670
C01514=1199.497,101.967,-49.988,-178.712,5.913,148.671
C01515=1199.502,101.717,-49.969,-178.714,5.912,148.671
C01516=1199.507,101.468,-49.950,-178.717,5.910,148.672
C01517=1199.512,101.219,-49.932,-178.720,5.910,148.672
C01518=1199.517,100.969,-49.913,-178.722,5.908,148.673
C01519=1199.522,100.720,-49.895,-178.725,5.907,148.673
C01520=1199.527,100.471,-49.877,-178.727,5.906,148.674
C01521=1199.531,100.222,-49.858,-178.730,5.905,148.675
C01522=1199.536,99.972,-49.839,-178.732,5.904,148.675
C01523=1199.541,99.723,-49.821,-178.736,5.903,148.676
C01524=1199.546,99.474,-49.803,-178.738,5.902,148.676
C01525=1199.551,99.224,-49.784,-178.740,5.901,148.677
C01526=1199.556,98.975,-49.766,-178.743,5.899,148.677
C01527=1199.560,98.727,-49.747,-178.746,5.899,148.678
C01528=1199.565,98.477,-49.729,-178.748,5.897,148.678
C01529=1199.570,98.227,-49.710,-178.751,5.896,148.679
C01530=1199.575,97.979,-49.691,-178.753,5.896,148.679
C01531=1199.580,97.729,-49.673,-178.756,5.894,148.680
C01532=1199.584,97.480,-49.655,-178.758,5.893,148.680
C01533=1199.590,97.230,-49.636,-178.761,5.893,148.681
C01534=1199.594,96.982,-49.618,-178.764,5.891,148.682
C01535=1199.599,96.732,-49.600,-178.766,5.890,148.682
C01536=1199.604,96.482,-49.581,-178.770,5.889,148.683
C01537=1199.608,96.233,-49.563,-178.772,5.888,148.683
C01538=1199.614,95.984,-49.545,-178.774,5.887,148.684
C01539=1199.619,95.735,-49.526,-178.777,5.886,148.684
C01540=1199.623,95.485,-49.508,-178.780,5.885,148.685
C01541=1199.628,95.236,-49.490,-178.782,5.884,148.685
C01542=1199.633,94.987,-49.472,-178.785,5.883,148.686
C01543=1199.638,94.738,-49.454,-178.787,5.882,148.686
C01544=1199.643,94.488,-49.435,-178.790,5.881,148.687
C01545=1199.648,94.238,-49.417,-178.792,5.880,148.687
C01546=1199.652,93.990,-49.398,-178.795,5.879,148.688
C01547=1199.657,93.741,-49.380,-178.798,5.877,148.688
C01548=1199.662,93.492,-49.362,-178.800,5.877,148.689
C01549=1199.667,93.242,-49.344,-178.803,5.876,148.690
C01550=1199.671,92.993,-49.326,-178.806,5.874,148.690
C01551=1199.677,92.743,-49.307,-178.808,5.874,148.691
C01552=1199.682,92.494,-49.289,-178.811,5.873,148.691
C01553=1199.687,92.245,-49.271,-178.814,5.871,148.692
C01554=1199.692,91.996,-49.253,-178.816,5.871,148.692
C01555=1199.697,91.746,-49.235,-178.819,5.869,148.693
C01556=1199.701,91.496,-49.217,-178.821,5.868,148.693
C01557=1199.706,91.247,-49.199,-178.824,5.868,148.694
C01558=1199.711,90.998,-49.181,-178.826,5.866,148.694
C01559=1199.716,90.749,-49.163,-178.829,5.865,148.695
C01560=1199.721,90.500,-49.145,-178.832,5.865,148.696
C01561=1199.726,90.251,-49.127,-178.834,5.863,148.696
C01562=1199.730,90.001,-49.109,-178.837,5.863,148.697
C01563=1199.735,89.752,-49.091,-178.839,5.862,148.697
C01564=1199.740,89.502,-49.073,-178.842,5.860,148.698
C01565=1199.745,89.253,-49.055,-178.845,5.859,148.698
C01566=1199.749,89.004,-49.037,-178.847,5.859,148.699
C01567=1199.754,88.755,-49.019,-178.850,5.857,148.699
C01568=1199.759,88.506,-49.001,-178.852,5.856,148.700
C01569=1199.764,88.256,-48.983,-178.855,5.856,148.701
C01570=1199.769,88.007,-48.965,-178.858,5.854,148.701
C01571=1199.774,87.757,-48.947,-178.860,5.854,148.702
C01572=1199.779,87.508,-48.929,-178.863,5.853,148.702
C01573=1199.784,87.258,-48.911,-178.866,5.851,148.703
C01574=1199.789,87.009,-48.893,-178.868,5.850,148.703
C01575=1199.793,86.760,-48.875,-178.871,5.850,148.704
C01576=1199.798,86.511,-48.857,-178.874,5.848,148.704
C01577=1199.803,86.262,-48.839,-178.876,5.847,148.705
C01578=1199.808,86.012,-48.822,-178.878,5.847,148.705
C01579=1199.813,85.763,-48.804,-178.881,5.846,148.706
C01580=1199.818,85.514,-48.786,-178.884,5.845,148.707
C01581=1199.823,85.264,-48.768,-178.886,5.844,148.707
C01582=1199.828,85.015,-48.750,-178.889,5.843,148.708
C01583=1199.833,84.765,-48.733,-178.892,5.842,148.708
C01584=1199.837,84.517,-48.716,-178.894,5.841,148.709
C01585=1199.842,84.267,-48.697,-178.897,5.840,148.709
C01586=1199.847,84.018,-48.679,-178.899,5.838,148.710
C01587=1199.852,83.768,-48.662,-178.902,5.838,148.710
C01588=1199.857,83.519,-48.644,-178.905,5.837,148.711
C01589=1199.862,83.269,-48.626,-178.907,5.836,148.711
C01590=1199.867,83.020,-48.608,-178.910,5.835,148.712
C01591=1199.872,82.770,-48.591,-178.912,5.834,148.713
C01592=1199.876,82.522,-48.573,-178.915,5.834,148.713
C01593=1199.881,82.272,-48.555,-178.917,5.832,148.714
C01594=1199.886,82.023,-48.538,-178.920,5.831,148.714
C01595=1199.891,81.773,-48.520,-178.923,5.831,148.715
C01596=1199.896,81.524,-48.502,-178.925,5.829,148.715
C01597=1199.901,81.255,-48.484,-178.928,5.828,148.716
C01598=1199.906,80.988,-48.465,-178.931,5.827,148.717
C01599=1199.912,80.719,-48.446,-178.934,5.826,148.717
C01600=1199.917,80.451,-48.427,-178.936,5.826,148.718
C01601=1199.922,80.201,-48.410,-178.939,5.824,148.718
C01602=1199.927,79.952,-48.392,-178.942,5.824,148.719
C01603=1199.932,79.702,-48.375,-178.944,5.823,148.719
C01604=1199.936,79.453,-48.357,-178.947,5.821,148.720
C01605=1199.941,79.204,-48.339,-178.949,5.820,148.721
C01606=1199.946,78.954,-48.322,-178.952,5.820,148.721
C01607=1199.951,78.705,-48.304,-178.954,5.819,148.722
C01608=1199.956,78.456,-48.287,-178.957,5.818,148.722
C01609=1199.961,78.207,-48.269,-178.960,5.817,148.723
C01610=1199.967,77.957,-48.252,-178.962,5.816,148.723
C01611=1199.972,77.708,-48.234,-178.965,5.815,148.724
C01612=1199.976,77.459,-48.218,-178.968,5.814,148.725
C01613=1199.981,77.210,-48.200,-178.970,5.813,148.725
C01614=1199.986,76.960,-48.182,-178.973,5.813,148.726
C01615=1199.990,76.711,-48.165,-178.976,5.811,148.726
C01616=1199.996,76.461,-48.148,-178.978,5.810,148.727
C01617=1200.000,76.212,-48.130,-178.980,5.810,148.727
C01618=1200.005,75.963,-48.113,-178.983,5.809,148.728
C01619=1200.010,75.713,-48.095,-178.986,5.808,148.729
C01620=1200.015,75.464,-48.078,-178.988,5.807,148.729
C01621=1200.020,75.214,-48.061,-178.991,5.806,148.730
C01622=1200.025,74.966,-48.044,-178.993,5.806,148.730
C01623=1200.030,74.716,-48.026,-178.996,5.804,148.731
C01624=1200.034,74.467,-48.009,-178.999,5.803,148.731
C01625=1200.040,74.217,-47.992,-179.001,5.803,148.732
C01626=1200.045,73.967,-47.974,-179.003,5.802,148.732
C01627=1200.049,73.718,-47.957,-179.007,5.800,148.733
C01628=1200.054,73.469,-47.940,-179.009,5.800,148.734
C01629=1200.059,73.220,-47.924,-179.011,5.799,148.734
C01630=1200.064,72.971,-47.906,-179.014,5.798,148.735
C01631=1200.069,72.721,-47.888,-179.017,5.797,148.736
C01632=1200.074,72.471,-47.872,-179.019,5.796,148.736
C01633=1200.079,72.222,-47.854,-179.022,5.796,148.737
C01634=1200.083,71.973,-47.837,-179.024,5.795,148.737
C01635=1200.089,71.723,-47.820,-179.027,5.793,148.738
C01636=1200.093,71.475,-47.803,-179.030,5.793,148.738
C01637=1200.099,71.225,-47.785,-179.032,5.792,148.739
C01638=1200.104,70.975,-47.768,-179.035,5.791,148.739
C01639=1200.108,70.726,-47.751,-179.037,5.791,148.740
C01640=1200.113,70.477,-47.733,-179.040,5.789,148.741
C01641=1200.118,70.228,-47.717,-179.043,5.788,148.741
C01642=1200.123,69.978,-47.700,-179.045,5.788,148.742
C01643=1200.128,69.728,-47.683,-179.047,5.787,148.742
C01644=1200.133,69.479,-47.665,-179.051,5.786,148.743
C01645=1200.137,69.230,-47.649,-179.053,5.785,148.744
C01646=1200.143,68.981,-47.632,-179.055,5.784,148.744
C01647=1200.148,68.731,-47.615,-179.058,5.784,148.745
C01648=1200.153,68.481,-47.598,-179.060,5.783,148.745
C01649=1200.157,68.233,-47.580,-179.063,5.781,148.746
C01650=1200.162,67.983,-47.563,-179.066,5.781,148.746
C01651=1200.167,67.734,-47.547,-179.068,5.780,148.747
C01652=1200.173,67.484,-47.530,-179.071,5.779,148.748
C01653=1200.177,67.235,-47.513,-179.074,5.778,148.748
C01654=1200.181,66.985,-47.496,-179.076,5.777,148.749
C01655=1200.187,66.736,-47.479,-179.079,5.776,148.749
C01656=1200.192,66.487,-47.463,-179.081,5.776,148.750
C01657=1200.197,66.238,-47.445,-179.084,5.775,148.750
C01658=1200.201,65.988,-47.428,-179.087,5.774,148.751
C01659=1200.207,65.739,-47.411,-179.089,5.773,148.752
C01660=1200.211,65.489,-47.394,-179.091,5.772,148.752
C01661=1200.216,65.240,-47.378,-179.094,5.772,148.753
C01662=1200.221,64.990,-47.360,-179.097,5.771,148.753
C01663=1200.226,64.741,-47.344,-179.099,5.769,148.754
C01664=1200.231,64.492,-47.327,-179.102,5.769,148.755
C01665=1200.236,64.242,-47.310,-179.105,5.768,148.755
C01666=1200.241,63.993,-47.294,-179.107,5.767,148.756
C01667=1200.246,63.744,-47.277,-179.110,5.767,148.756
C01668=1200.251,63.494,-47.260,-179.112,5.766,148.757
C01669=1200.255,63.245,-47.243,-179.115,5.765,148.757
C01670=1200.261,62.995,-47.226,-179.118,5.764,148.758
C01671=1200.266,62.746,-47.210,-179.120,5.763,148.759
C01672=1200.270,62.496,-47.193,-179.122,5.763,148.759
C01673=1200.276,62.247,-47.176,-179.125,5.762,148.760
C01674=1200.280,61.998,-47.160,-179.128,5.761,148.760
C01675=1200.285,61.748,-47.143,-179.130,5.760,148.761
C01676=1200.291,61.499,-47.126,-179.133,5.759,148.762
C01677=1200.295,61.250,-47.109,-179.136,5.759,148.762
C01678=1200.300,61.000,-47.093,-179.138,5.758,148.763
C01679=1200.306,60.751,-47.076,-179.140,5.757,148.763
C01680=1200.310,60.501,-47.060,-179.144,5.756,148.764
C01681=1200.315,60.252,-47.043,-179.146,5.755,148.764
C01682=1200.320,60.003,-47.027,-179.148,5.754,148.765
C01683=1200.325,59.753,-47.010,-179.151,5.754,148.766
C01684=1200.329,59.504,-46.993,-179.154,5.753,148.766
C01685=1200.334,59.255,-46.977,-179.156,5.752,148.767
C01686=1200.339,59.005,-46.961,-179.159,5.751,148.768
C01687=1200.345,58.756,-46.944,-179.162,5.751,148.768
C01688=1200.350,58.506,-46.927,-179.164,5.750,148.769
C01689=1200.354,58.257,-46.910,-179.166,5.749,148.769
C01690=1200.359,58.008,-46.894,-179.169,5.749,148.770
C01691=1200.364,57.758,-46.877,-179.171,5.748,148.770
C01692=1200.370,57.509,-46.861,-179.174,5.746,148.771
C01693=1200.374,57.259,-46.845,-179.177,5.746,148.772
C01694=1200.379,57.010,-46.828,-179.179,5.745,148.772
C01695=1200.385,56.761,-46.811,-179.182,5.744,148.773
C01696=1200.389,56.511,-46.795,-179.184,5.744,148.774
C01697=1200.394,56.262,-46.779,-179.187,5.743,148.774
C01698=1200.399,56.012,-46.762,-179.190,5.741,148.775
C01699=1200.403,55.763,-46.745,-179.192,5.741,148.775
C01700=1200.409,55.513,-46.730,-179.195,5.740,148.776
C01701=1200.415,55.245,-46.711,-179.198,5.740,148.777
C01702=1200.420,54.976,-46.694,-179.200,5.739,148.777
C01703=1200.425,54.708,-46.676,-179.203,5.738,148.778
C01704=1200.430,54.439,-46.659,-179.206,5.737,148.778
C01705=1200.435,54.190,-46.643,-179.208,5.737,148.779
C01706=1200.439,53.941,-46.626,-179.211,5.736,148.780
C01707=1200.446,53.691,-46.610,-179.213,5.735,148.780
C01708=1200.450,53.442,-46.593,-179.216,5.734,148.781
C01709=1200.455,53.192,-46.578,-179.219,5.733,148.781
C01710=1200.460,52.943,-46.561,-179.221,5.732,148.782
C01711=1200.465,52.694,-46.545,-179.224,5.732,148.783
C01712=1200.470,52.444,-46.529,-179.226,5.731,148.783
C01713=1200.475,52.195,-46.512,-179.229,5.731,148.784
C01714=1200.479,51.945,-46.496,-179.231,5.730,148.784
C01715=1200.485,51.696,-46.480,-179.234,5.729,148.785
C01716=1200.489,51.447,-46.463,-179.237,5.728,148.786
C01717=1200.495,51.197,-46.448,-179.239,5.727,148.786
C01718=1200.499,50.948,-46.431,-179.242,5.726,148.787
C01719=1200.505,50.698,-46.415,-179.244,5.726,148.787
C01720=1200.510,50.449,-46.398,-179.247,5.725,148.788
C01721=1200.515,50.199,-46.383,-179.249,5.724,148.789
C01722=1200.520,49.950,-46.366,-179.252,5.724,148.789
C01723=1200.525,49.700,-46.350,-179.254,5.723,148.790
C01724=1200.529,49.451,-46.334,-179.257,5.722,148.790
C01725=1200.535,49.201,-46.318,-179.260,5.721,148.791
C01726=1200.539,48.952,-46.302,-179.262,5.721,148.792
C01727=1200.545,48.702,-46.286,-179.265,5.720,148.792
C01728=1200.549,48.453,-46.269,-179.267,5.719,148.793
C01729=1200.555,48.204,-46.254,-179.270,5.719,148.793
C01730=1200.559,47.954,-46.237,-179.273,5.718,148.794
C01731=1200.564,47.705,-46.221,-179.275,5.718,148.795
C01732=1200.569,47.455,-46.205,-179.277,5.717,148.795
C01733=1200.574,47.206,-46.190,-179.280,5.716,148.796
C01734=1200.579,46.957,-46.174,-179.283,5.715,148.797
C01735=1200.583,46.707,-46.158,-179.285,5.714,148.797
C01736=1200.589,46.458,-46.142,-179.288,5.713,148.798
C01737=1200.593,46.208,-46.125,-179.291,5.713,148.798
C01738=1200.599,45.959,-46.110,-179.293,5.712,148.799
C01739=1200.603,45.709,-46.094,-179.295,5.711,148.800
C01740=1200.609,45.460,-46.077,-179.298,5.711,148.800
C01741=1200.614,45.211,-46.062,-179.301,5.710,148.801
C01742=1200.619,44.961,-46.046,-179.303,5.710,148.802
C01743=1200.624,44.712,-46.030,-179.305,5.709,148.802
C01744=1200.629,44.462,-46.014,-179.308,5.708,148.803
C01745=1200.634,44.212,-45.998,-179.311,5.707,148.803
C01746=1200.638,43.964,-45.982,-179.314,5.707,148.804
C01747=1200.643,43.714,-45.966,-179.316,5.706,148.804
C01748=1200.648,43.464,-45.951,-179.319,5.705,148.805
C01749=1200.654,43.215,-45.934,-179.321,5.705,148.806
C01750=1200.658,42.965,-45.919,-179.324,5.704,148.806
C01751=1200.664,42.716,-45.903,-179.326,5.703,148.807
C01752=1200.669,42.466,-45.887,-179.329,5.703,148.808
C01753=1200.673,42.217,-45.871,-179.331,5.702,148.808
C01754=1200.678,41.968,-45.856,-179.334,5.701,148.809
C01755=1200.683,41.718,-45.840,-179.336,5.701,148.809
C01756=1200.688,41.468,-45.824,-179.339,5.700,148.810
C01757=1200.693,41.220,-45.808,-179.342,5.700,148.811
C01758=1200.698,40.970,-45.792,-179.344,5.698,148.811
C01759=1200.703,40.721,-45.777,-179.347,5.697,148.812
C01760=1200.708,40.471,-45.761,-179.350,5.697,148.812
C01761=1200.713,40.221,-45.745,-179.352,5.696,148.813
C01762=1200.718,39.972,-45.729,-179.354,5.695,148.814
C01763=1200.724,39.723,-45.713,-179.357,5.695,148.814
C01764=1200.728,39.473,-45.698,-179.360,5.694,148.815
C01765=1200.733,39.224,-45.683,-179.362,5.694,148.816
C01766=1200.738,38.974,-45.667,-179.364,5.693,148.816
C01767=1200.744,38.725,-45.651,-179.367,5.692,148.817
C01768=1200.748,38.475,-45.636,-179.370,5.692,148.817
C01769=1200.753,38.226,-45.620,-179.372,5.691,148.818
C01770=1200.758,37.977,-45.604,-179.374,5.691,148.819
C01771=1200.763,37.727,-45.588,-179.377,5.690,148.819
C01772=1200.768,37.478,-45.573,-179.380,5.689,148.820
C01773=1200.773,37.228,-45.558,-179.382,5.689,148.821
C01774=1200.779,36.979,-45.542,-179.385,5.688,148.821
C01775=1200.783,36.729,-45.527,-179.388,5.687,148.822
C01776=1200.788,36.480,-45.511,-179.390,5.686,148.822
C01777=1200.793,36.230,-45.495,-179.393,5.686,148.823
C01778=1200.798,35.980,-45.479,-179.395,5.685,148.823
C01779=1200.803,35.731,-45.464,-179.398,5.684,148.824
C01780=1200.808,35.482,-45.449,-179.401,5.684,148.825
C01781=1200.814,35.232,-45.433,-179.403,5.683,148.825
C01782=1200.818,34.982,-45.418,-179.406,5.683,148.826
C01783=1200.823,34.733,-45.402,-179.408,5.682,148.827
C01784=1200.828,34.484,-45.387,-179.411,5.681,148.827
C01785=1200.833,34.235,-45.372,-179.413,5.681,148.828
C01786=1200.838,33.985,-45.356,-179.416,5.680,148.829
C01787=1200.843,33.735,-45.340,-179.418,5.679,148.829
C01788=1200.848,33.486,-45.325,-179.421,5.679,148.830
C01789=1200.853,33.237,-45.310,-179.423,5.678,148.830
C01790=1200.858,32.987,-45.295,-179.426,5.678,148.831
C01791=1200.863,32.737,-45.279,-179.428,5.677,148.832
C01792=1200.868,32.488,-45.263,-179.431,5.676,148.832
C01793=1200.873,32.239,-45.248,-179.433,5.676,148.833
C01794=1200.878,31.989,-45.233,-179.436,5.675,148.834
C01795=1200.883,31.740,-45.218,-179.439,5.675,148.834
C01796=1200.888,31.490,-45.202,-179.441,5.674,148.835
C01797=1200.893,31.240,-45.187,-179.443,5.673,148.835
C01798=1200.898,30.991,-45.172,-179.446,5.673,148.836
C01799=1200.903,30.742,-45.156,-179.449,5.672,148.837
C01800=1200.908,30.493,-45.141,-179.451,5.671,148.837
C01801=1200.913,30.243,-45.126,-179.454,5.671,148.838
C01802=1200.918,29.993,-45.111,-179.456,5.670,148.839
C01803=1200.923,29.743,-45.095,-179.459,5.670,148.839
C01804=1200.928,29.494,-45.080,-179.461,5.669,148.840
C01805=1200.934,29.225,-45.064,-179.464,5.669,148.840
C01806=1200.939,28.957,-45.047,-179.467,5.667,148.841
C01807=1200.944,28.688,-45.031,-179.470,5.667,148.842
C01808=1200.950,28.420,-45.014,-179.472,5.666,148.842
C01809=1200.954,28.170,-44.999,-179.475,5.666,148.843
C01810=1200.960,27.920,-44.984,-179.477,5.665,148.844
C01811=1200.964,27.671,-44.969,-179.480,5.665,148.844
C01812=1200.970,27.421,-44.953,-179.483,5.664,148.845
C01813=1200.974,27.172,-44.938,-179.485,5.663,148.846
C01814=1200.980,26.922,-44.924,-179.488,5.663,148.846
